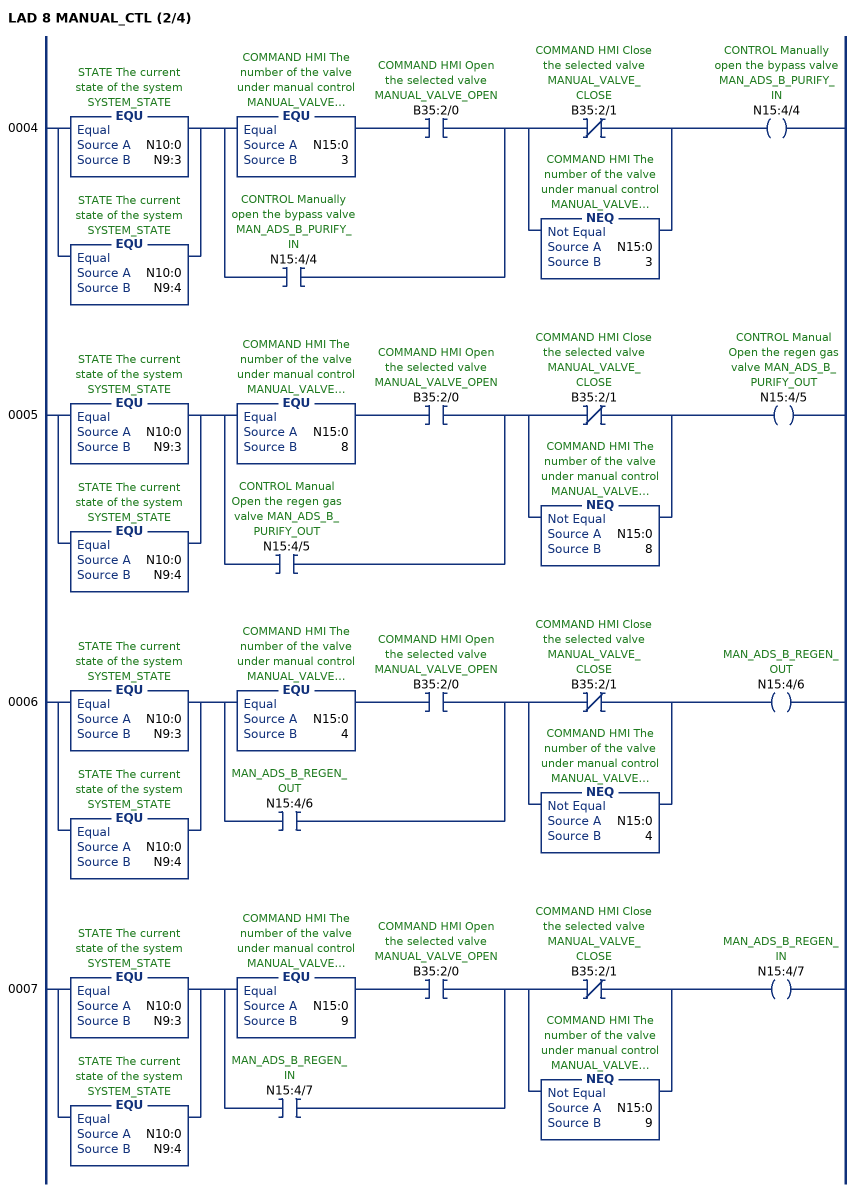
% Rung: 4 %
SOR BST EQU N10:0 N9:3 NXB EQU N10:0 N9:4 BND BST EQU N15:0 3 XIC B35:2/0 NXB XIC N15:4/4 BND BST XIO B35:2/1 NXB NEQ N15:0 3 BND OTE N15:4/4 EOR
%   N10:0  SYSTEM_STATE  "STATE The current state of the system" %
%   N9:3  SYSTEM_MANUAL  "STATE System Manual" %
%   N9:4  SYSTEM_ALARM  "STATE System Alarm" %
%   N15:0  MANUAL_VALVE_NUMBER  "COMMAND HMI The number of the valve under manual control" %
%   B35:2/0  MANUAL_VALVE_OPEN  "COMMAND HMI Open the selected valve" %
%   N15:4/4  MAN_ADS_B_PURIFY_IN  "CONTROL Manually open the bypass valve" %
%   B35:2/1  MANUAL_VALVE_CLOSE  "COMMAND HMI Close the selected valve" %
% Rung: 5 %
SOR BST EQU N10:0 N9:3 NXB EQU N10:0 N9:4 BND BST EQU N15:0 8 XIC B35:2/0 NXB XIC N15:4/5 BND BST XIO B35:2/1 NXB NEQ N15:0 8 BND OTE N15:4/5 EOR
%   N10:0  SYSTEM_STATE  "STATE The current state of the system" %
%   N9:3  SYSTEM_MANUAL  "STATE System Manual" %
%   N9:4  SYSTEM_ALARM  "STATE System Alarm" %
%   N15:0  MANUAL_VALVE_NUMBER  "COMMAND HMI The number of the valve under manual control" %
%   B35:2/0  MANUAL_VALVE_OPEN  "COMMAND HMI Open the selected valve" %
%   N15:4/5  MAN_ADS_B_PURIFY_OUT  "CONTROL Manual Open the regen gas valve" %
%   B35:2/1  MANUAL_VALVE_CLOSE  "COMMAND HMI Close the selected valve" %
% Rung: 6 %
SOR BST EQU N10:0 N9:3 NXB EQU N10:0 N9:4 BND BST EQU N15:0 4 XIC B35:2/0 NXB XIC N15:4/6 BND BST XIO B35:2/1 NXB NEQ N15:0 4 BND OTE N15:4/6 EOR
%   N10:0  SYSTEM_STATE  "STATE The current state of the system" %
%   N9:3  SYSTEM_MANUAL  "STATE System Manual" %
%   N9:4  SYSTEM_ALARM  "STATE System Alarm" %
%   N15:0  MANUAL_VALVE_NUMBER  "COMMAND HMI The number of the valve under manual control" %
%   B35:2/0  MANUAL_VALVE_OPEN  "COMMAND HMI Open the selected valve" %
%   N15:4/6  MAN_ADS_B_REGEN_OUT %
%   B35:2/1  MANUAL_VALVE_CLOSE  "COMMAND HMI Close the selected valve" %
% Rung: 7 %
SOR BST EQU N10:0 N9:3 NXB EQU N10:0 N9:4 BND BST EQU N15:0 9 XIC B35:2/0 NXB XIC N15:4/7 BND BST XIO B35:2/1 NXB NEQ N15:0 9 BND OTE N15:4/7 EOR
%   N10:0  SYSTEM_STATE  "STATE The current state of the system" %
%   N9:3  SYSTEM_MANUAL  "STATE System Manual" %
%   N9:4  SYSTEM_ALARM  "STATE System Alarm" %
%   N15:0  MANUAL_VALVE_NUMBER  "COMMAND HMI The number of the valve under manual control" %
%   B35:2/0  MANUAL_VALVE_OPEN  "COMMAND HMI Open the selected valve" %
%   N15:4/7  MAN_ADS_B_REGEN_IN %
%   B35:2/1  MANUAL_VALVE_CLOSE  "COMMAND HMI Close the selected valve" %

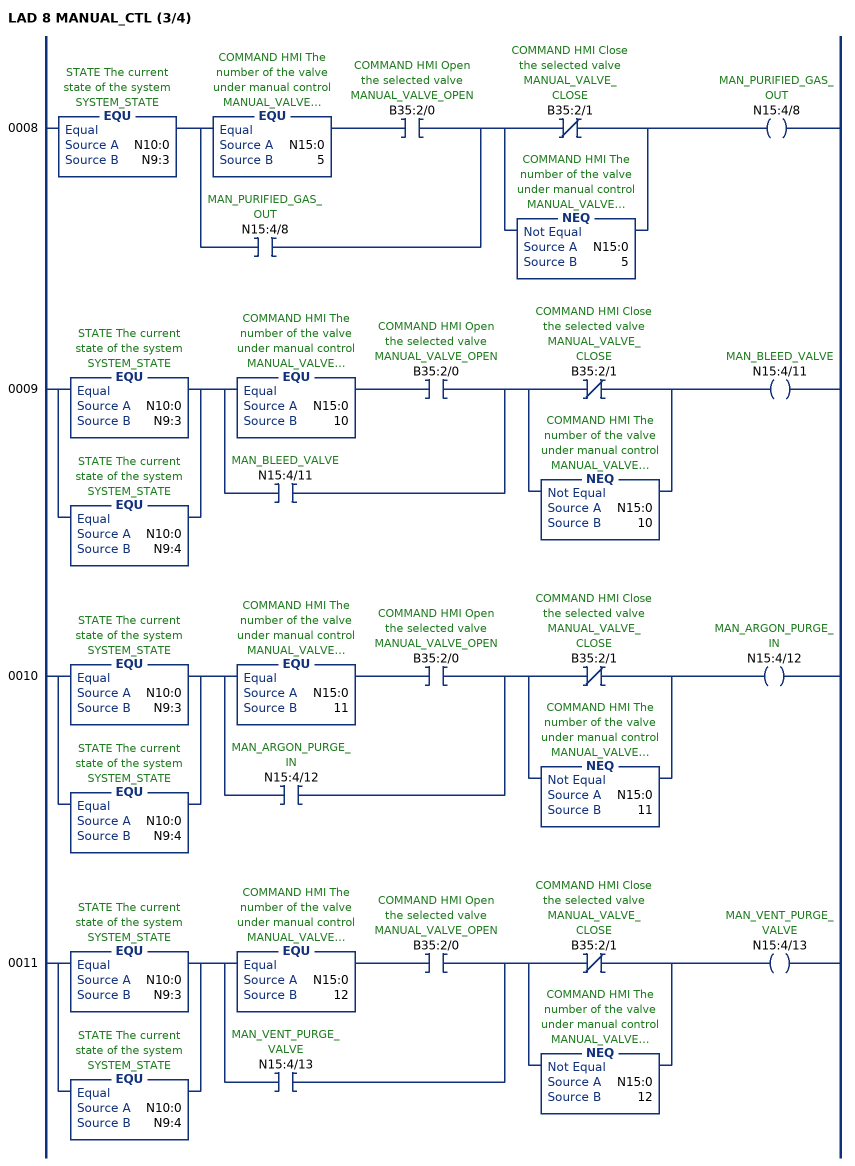
% Rung: 8 %
SOR EQU N10:0 N9:3 BST EQU N15:0 5 XIC B35:2/0 NXB XIC N15:4/8 BND BST XIO B35:2/1 NXB NEQ N15:0 5 BND OTE N15:4/8 EOR
%   N10:0  SYSTEM_STATE  "STATE The current state of the system" %
%   N9:3  SYSTEM_MANUAL  "STATE System Manual" %
%   N15:0  MANUAL_VALVE_NUMBER  "COMMAND HMI The number of the valve under manual control" %
%   B35:2/0  MANUAL_VALVE_OPEN  "COMMAND HMI Open the selected valve" %
%   N15:4/8  MAN_PURIFIED_GAS_OUT %
%   B35:2/1  MANUAL_VALVE_CLOSE  "COMMAND HMI Close the selected valve" %
% Rung: 9 %
SOR BST EQU N10:0 N9:3 NXB EQU N10:0 N9:4 BND BST EQU N15:0 10 XIC B35:2/0 NXB XIC N15:4/11 BND BST XIO B35:2/1 NXB NEQ N15:0 10 BND OTE N15:4/11 EOR
%   N10:0  SYSTEM_STATE  "STATE The current state of the system" %
%   N9:3  SYSTEM_MANUAL  "STATE System Manual" %
%   N9:4  SYSTEM_ALARM  "STATE System Alarm" %
%   N15:0  MANUAL_VALVE_NUMBER  "COMMAND HMI The number of the valve under manual control" %
%   B35:2/0  MANUAL_VALVE_OPEN  "COMMAND HMI Open the selected valve" %
%   N15:4/11  MAN_BLEED_VALVE %
%   B35:2/1  MANUAL_VALVE_CLOSE  "COMMAND HMI Close the selected valve" %
% Rung: 10 %
SOR BST EQU N10:0 N9:3 NXB EQU N10:0 N9:4 BND BST EQU N15:0 11 XIC B35:2/0 NXB XIC N15:4/12 BND BST XIO B35:2/1 NXB NEQ N15:0 11 BND OTE N15:4/12 EOR
%   N10:0  SYSTEM_STATE  "STATE The current state of the system" %
%   N9:3  SYSTEM_MANUAL  "STATE System Manual" %
%   N9:4  SYSTEM_ALARM  "STATE System Alarm" %
%   N15:0  MANUAL_VALVE_NUMBER  "COMMAND HMI The number of the valve under manual control" %
%   B35:2/0  MANUAL_VALVE_OPEN  "COMMAND HMI Open the selected valve" %
%   N15:4/12  MAN_ARGON_PURGE_IN %
%   B35:2/1  MANUAL_VALVE_CLOSE  "COMMAND HMI Close the selected valve" %
% Rung: 11 %
SOR BST EQU N10:0 N9:3 NXB EQU N10:0 N9:4 BND BST EQU N15:0 12 XIC B35:2/0 NXB XIC N15:4/13 BND BST XIO B35:2/1 NXB NEQ N15:0 12 BND OTE N15:4/13 EOR
%   N10:0  SYSTEM_STATE  "STATE The current state of the system" %
%   N9:3  SYSTEM_MANUAL  "STATE System Manual" %
%   N9:4  SYSTEM_ALARM  "STATE System Alarm" %
%   N15:0  MANUAL_VALVE_NUMBER  "COMMAND HMI The number of the valve under manual control" %
%   B35:2/0  MANUAL_VALVE_OPEN  "COMMAND HMI Open the selected valve" %
%   N15:4/13  MAN_VENT_PURGE_VALVE %
%   B35:2/1  MANUAL_VALVE_CLOSE  "COMMAND HMI Close the selected valve" %

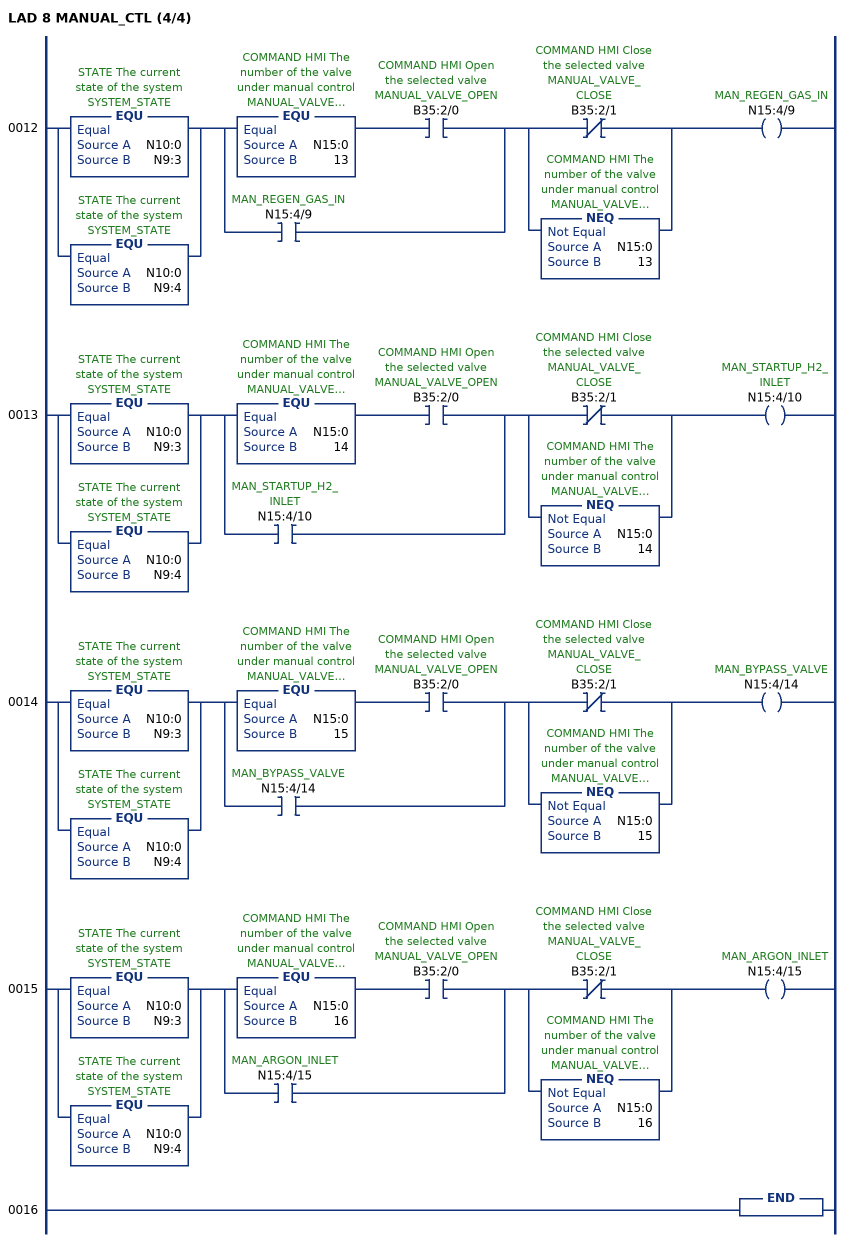
% Rung: 12 %
SOR BST EQU N10:0 N9:3 NXB EQU N10:0 N9:4 BND BST EQU N15:0 13 XIC B35:2/0 NXB XIC N15:4/9 BND BST XIO B35:2/1 NXB NEQ N15:0 13 BND OTE N15:4/9 EOR
%   N10:0  SYSTEM_STATE  "STATE The current state of the system" %
%   N9:3  SYSTEM_MANUAL  "STATE System Manual" %
%   N9:4  SYSTEM_ALARM  "STATE System Alarm" %
%   N15:0  MANUAL_VALVE_NUMBER  "COMMAND HMI The number of the valve under manual control" %
%   B35:2/0  MANUAL_VALVE_OPEN  "COMMAND HMI Open the selected valve" %
%   N15:4/9  MAN_REGEN_GAS_IN %
%   B35:2/1  MANUAL_VALVE_CLOSE  "COMMAND HMI Close the selected valve" %
% Rung: 13 %
SOR BST EQU N10:0 N9:3 NXB EQU N10:0 N9:4 BND BST EQU N15:0 14 XIC B35:2/0 NXB XIC N15:4/10 BND BST XIO B35:2/1 NXB NEQ N15:0 14 BND OTE N15:4/10 EOR
%   N10:0  SYSTEM_STATE  "STATE The current state of the system" %
%   N9:3  SYSTEM_MANUAL  "STATE System Manual" %
%   N9:4  SYSTEM_ALARM  "STATE System Alarm" %
%   N15:0  MANUAL_VALVE_NUMBER  "COMMAND HMI The number of the valve under manual control" %
%   B35:2/0  MANUAL_VALVE_OPEN  "COMMAND HMI Open the selected valve" %
%   N15:4/10  MAN_STARTUP_H2_INLET %
%   B35:2/1  MANUAL_VALVE_CLOSE  "COMMAND HMI Close the selected valve" %
% Rung: 14 %
SOR BST EQU N10:0 N9:3 NXB EQU N10:0 N9:4 BND BST EQU N15:0 15 XIC B35:2/0 NXB XIC N15:4/14 BND BST XIO B35:2/1 NXB NEQ N15:0 15 BND OTE N15:4/14 EOR
%   N10:0  SYSTEM_STATE  "STATE The current state of the system" %
%   N9:3  SYSTEM_MANUAL  "STATE System Manual" %
%   N9:4  SYSTEM_ALARM  "STATE System Alarm" %
%   N15:0  MANUAL_VALVE_NUMBER  "COMMAND HMI The number of the valve under manual control" %
%   B35:2/0  MANUAL_VALVE_OPEN  "COMMAND HMI Open the selected valve" %
%   N15:4/14  MAN_BYPASS_VALVE %
%   B35:2/1  MANUAL_VALVE_CLOSE  "COMMAND HMI Close the selected valve" %
% Rung: 15 %
SOR BST EQU N10:0 N9:3 NXB EQU N10:0 N9:4 BND BST EQU N15:0 16 XIC B35:2/0 NXB XIC N15:4/15 BND BST XIO B35:2/1 NXB NEQ N15:0 16 BND OTE N15:4/15 EOR
%   N10:0  SYSTEM_STATE  "STATE The current state of the system" %
%   N9:3  SYSTEM_MANUAL  "STATE System Manual" %
%   N9:4  SYSTEM_ALARM  "STATE System Alarm" %
%   N15:0  MANUAL_VALVE_NUMBER  "COMMAND HMI The number of the valve under manual control" %
%   B35:2/0  MANUAL_VALVE_OPEN  "COMMAND HMI Open the selected valve" %
%   N15:4/15  MAN_ARGON_INLET %
%   B35:2/1  MANUAL_VALVE_CLOSE  "COMMAND HMI Close the selected valve" %
% Rung: 16 %
SOR END EOR

LADDER 9 "STARTUP"
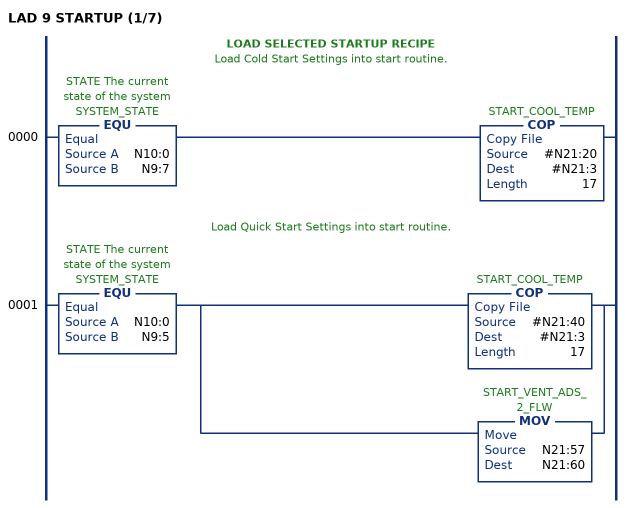
% Rung: 0 %
% TITLE: LOAD SELECTED STARTUP RECIPE %
% Load Cold Start Settings into start routine. %
SOR EQU N10:0 N9:7 COP #N21:20 #N21:3 17 EOR
%   N10:0  SYSTEM_STATE  "STATE The current state of the system" %
%   N9:7  SYSTEM_COLD_START %
%   N21:20  COLD_COOL_TEMP %
%   N21:3  START_COOL_TEMP %
% Rung: 1 %
% Load Quick Start Settings into start routine. %
SOR EQU N10:0 N9:5 BST COP #N21:40 #N21:3 17 NXB MOV N21:57 N21:60 BND EOR
%   N10:0  SYSTEM_STATE  "STATE The current state of the system" %
%   N9:5  SYSTEM_QUICK_START %
%   N21:40  QUICK_COOL_TEMP %
%   N21:3  START_COOL_TEMP %
%   N21:57  QUICK_VENT_ADS_2_FLW %
%   N21:60  START_VENT_ADS_2_FLW %

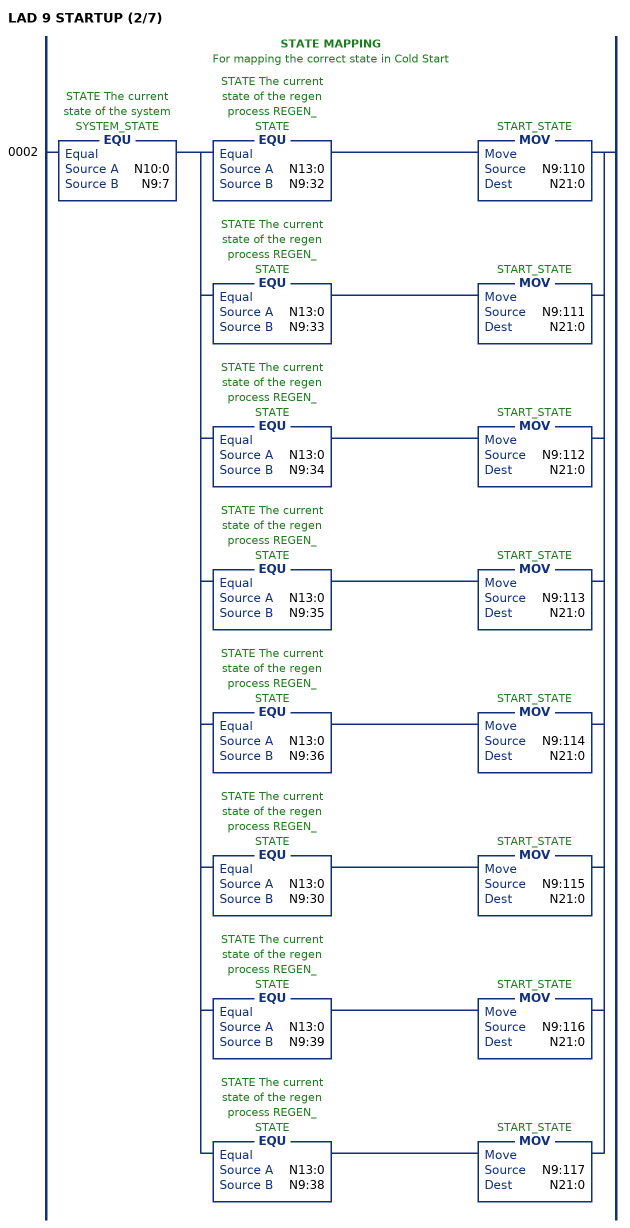
% Rung: 2 %
% TITLE: STATE MAPPING %
% For mapping the correct state in Cold Start %
SOR EQU N10:0 N9:7 BST EQU N13:0 N9:32 MOV N9:110 N21:0 NXB EQU N13:0 N9:33 MOV N9:111 N21:0 NXB EQU N13:0 N9:34 MOV N9:112 N21:0 NXB EQU N13:0 N9:35 MOV N9:113 N21:0 NXB EQU N13:0 N9:36 MOV N9:114 N21:0 NXB EQU N13:0 N9:30 MOV N9:115 N21:0 NXB EQU N13:0 N9:39 MOV N9:116 N21:0 NXB EQU N13:0 N9:38 MOV N9:117 N21:0 BND EOR
%   N10:0  SYSTEM_STATE  "STATE The current state of the system" %
%   N9:7  SYSTEM_COLD_START %
%   N13:0  REGEN_STATE  "STATE The current state of the regen process" %
%   N9:32  REGEN_VENT  "STATE Regen Vent" %
%   N9:110  START_REG_VENT %
%   N21:0  START_STATE %
%   N9:33  REGEN_HEAT_BED  "STATE Regen Heat wall" %
%   N9:111  START_REG_HEAT %
%   N9:34  REGEN_RUN  "STATE Regen Running" %
%   N9:112  START_REG_RUN %
%   N9:35  REGEN_COOL_WALL  "STATE Regen Cool wall" %
%   N9:113  START_REG_COOL %
%   N9:36  REGEN_COOL  "STATE Regen Cool" %
%   N9:114  START_REG_TIMED_COOL %
%   N9:30  REGEN_STANDBY  "STATE Regen Standby" %
%   N9:115  START_REG_STANDBY %
%   N9:39  REGEN_BACKFILL %
%   N9:116  START_REG_BACKFILL %
%   N9:38  REGEN_DONE %
%   N9:117  START_REG_DONE %

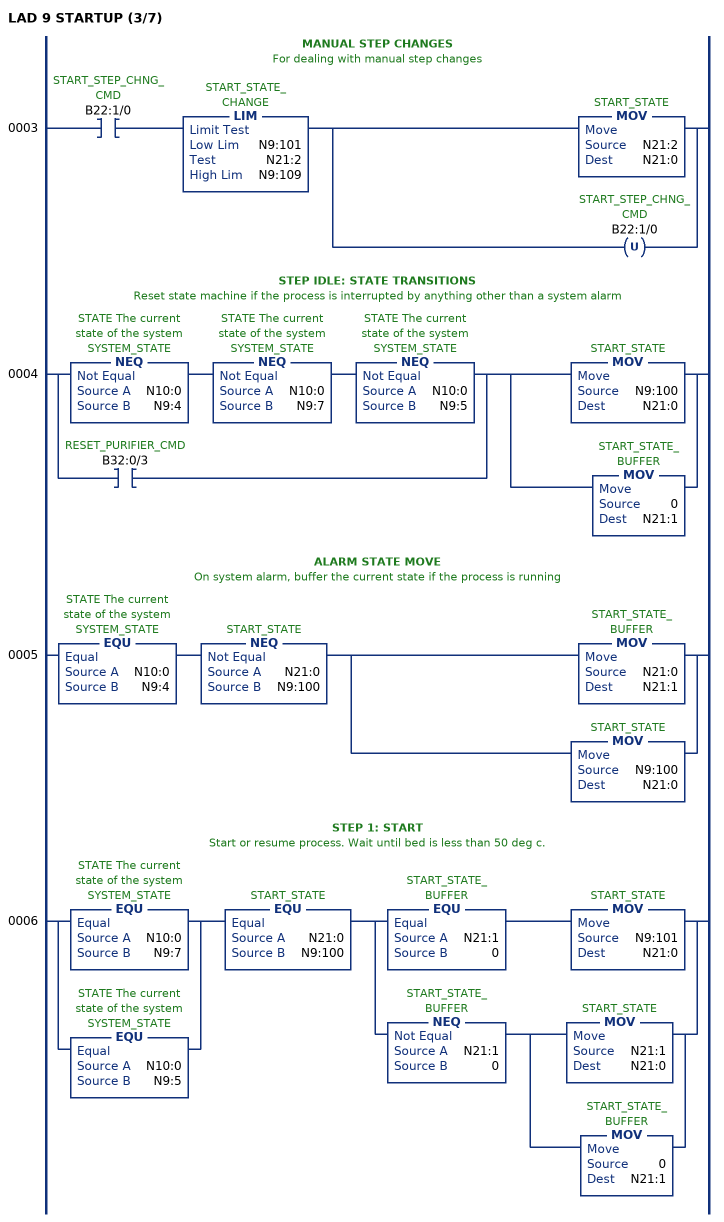
% Rung: 3 %
% TITLE: MANUAL STEP CHANGES %
% For dealing with manual step changes %
SOR XIC B22:1/0 LIM N9:101 N21:2 N9:109 BST MOV N21:2 N21:0 NXB OTU B22:1/0 BND EOR
%   B22:1/0  START_STEP_CHNG_CMD %
%   N9:101  START_COOL %
%   N21:2  START_STATE_CHANGE %
%   N9:109  START_BKFL_2 %
%   N21:0  START_STATE %
% Rung: 4 %
% TITLE: STEP IDLE: STATE TRANSITIONS %
% Reset state machine if the process is interrupted by anything other than a system alarm %
SOR BST NEQ N10:0 N9:4 NEQ N10:0 N9:7 NEQ N10:0 N9:5 NXB XIC B32:0/3 BND BST MOV N9:100 N21:0 NXB MOV 0 N21:1 BND EOR
%   N10:0  SYSTEM_STATE  "STATE The current state of the system" %
%   N9:4  SYSTEM_ALARM  "STATE System Alarm" %
%   N9:7  SYSTEM_COLD_START %
%   N9:5  SYSTEM_QUICK_START %
%   B32:0/3  RESET_PURIFIER_CMD %
%   N9:100  START_IDLE %
%   N21:0  START_STATE %
%   N21:1  START_STATE_BUFFER %
% Rung: 5 %
% TITLE: ALARM STATE MOVE %
% On system alarm, buffer the current state if the process is running %
SOR EQU N10:0 N9:4 NEQ N21:0 N9:100 BST MOV N21:0 N21:1 NXB MOV N9:100 N21:0 BND EOR
%   N10:0  SYSTEM_STATE  "STATE The current state of the system" %
%   N9:4  SYSTEM_ALARM  "STATE System Alarm" %
%   N21:0  START_STATE %
%   N9:100  START_IDLE %
%   N21:1  START_STATE_BUFFER %
% Rung: 6 %
% TITLE: STEP 1: START %
% Start or resume process. Wait until bed is less than 50 deg c. %
SOR BST EQU N10:0 N9:7 NXB EQU N10:0 N9:5 BND EQU N21:0 N9:100 BST EQU N21:1 0 MOV N9:101 N21:0 NXB NEQ N21:1 0 BST MOV N21:1 N21:0 NXB MOV 0 N21:1 BND BND EOR
%   N10:0  SYSTEM_STATE  "STATE The current state of the system" %
%   N9:7  SYSTEM_COLD_START %
%   N9:5  SYSTEM_QUICK_START %
%   N21:0  START_STATE %
%   N9:100  START_IDLE %
%   N21:1  START_STATE_BUFFER %
%   N9:101  START_COOL %

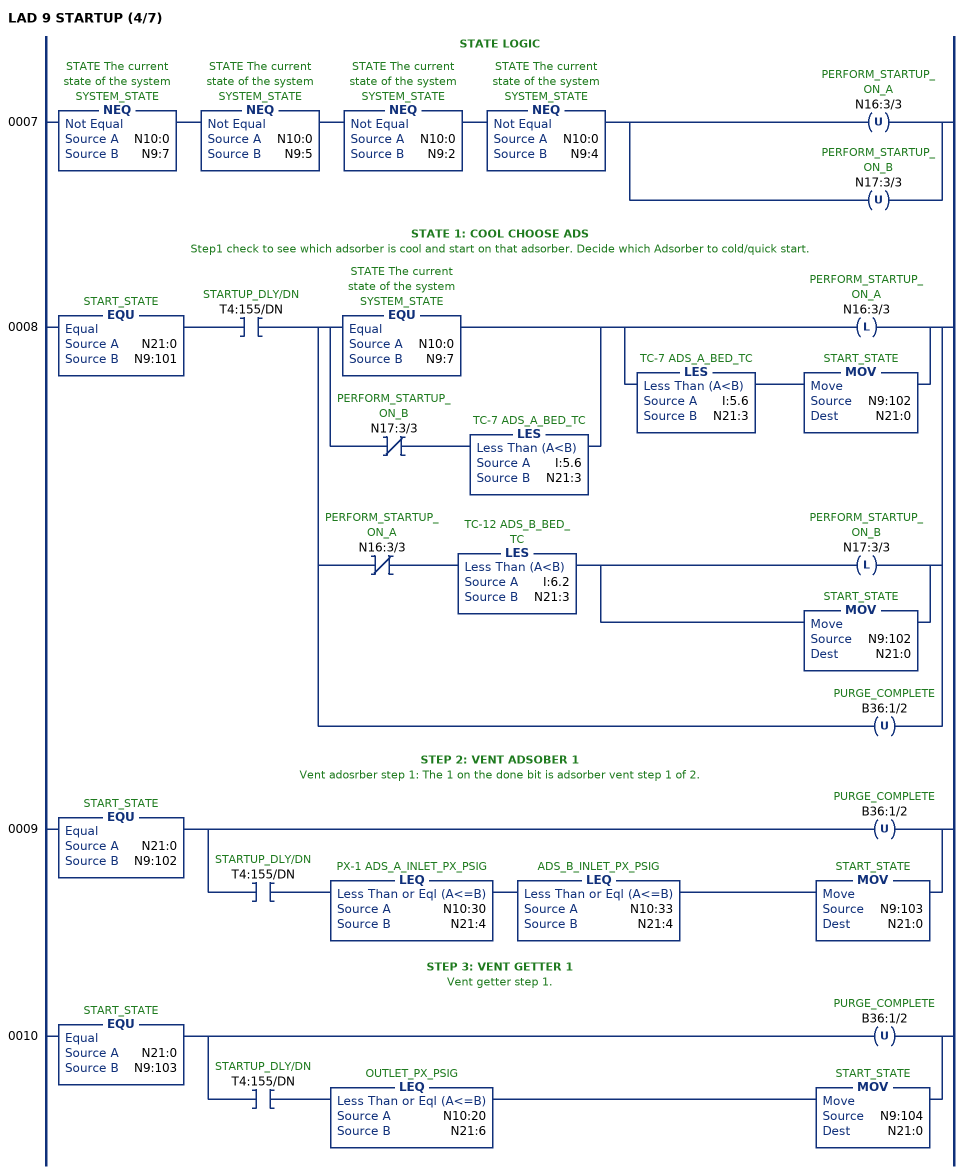
% Rung: 7 %
% TITLE: STATE LOGIC %
SOR NEQ N10:0 N9:7 NEQ N10:0 N9:5 NEQ N10:0 N9:2 NEQ N10:0 N9:4 BST OTU N16:3/3 NXB OTU N17:3/3 BND EOR
%   N10:0  SYSTEM_STATE  "STATE The current state of the system" %
%   N9:7  SYSTEM_COLD_START %
%   N9:5  SYSTEM_QUICK_START %
%   N9:2  SYSTEM_PROCESS  "STATE System Process" %
%   N9:4  SYSTEM_ALARM  "STATE System Alarm" %
%   N16:3/3  PERFORM_STARTUP_ON_A %
%   N17:3/3  PERFORM_STARTUP_ON_B %
% Rung: 8 %
% TITLE: STATE 1: COOL CHOOSE ADS %
% Step1 check to see which adsorber is cool and start on that adsorber. Decide which Adsorber to cold/quick start. %
SOR EQU N21:0 N9:101 XIC T4:155/DN BST BST EQU N10:0 N9:7 NXB XIO N17:3/3 LES I:5.6 N21:3 BND BST OTL N16:3/3 NXB LES I:5.6 N21:3 MOV N9:102 N21:0 BND NXB XIO N16:3/3 LES I:6.2 N21:3 BST OTL N17:3/3 NXB MOV N9:102 N21:0 BND NXB OTU B36:1/2 BND EOR
%   N21:0  START_STATE %
%   N9:101  START_COOL %
%   T4:155  STARTUP_DLY %
%   N10:0  SYSTEM_STATE  "STATE The current state of the system" %
%   N9:7  SYSTEM_COLD_START %
%   N17:3/3  PERFORM_STARTUP_ON_B %
%   I:5.6  ADS_A_BED_TC  "TC-7" %
%   N21:3  START_COOL_TEMP %
%   N16:3/3  PERFORM_STARTUP_ON_A %
%   N9:102  START_VENT_ADS_1 %
%   I:6.2  ADS_B_BED_TC  "TC-12" %
%   B36:1/2  PURGE_COMPLETE %
% Rung: 9 %
% TITLE: STEP 2: VENT ADSOBER 1 %
% Vent adosrber step 1: The 1 on the done bit is adsorber vent step 1 of 2. %
SOR EQU N21:0 N9:102 BST OTU B36:1/2 NXB XIC T4:155/DN LEQ N10:30 N21:4 LEQ N10:33 N21:4 MOV N9:103 N21:0 BND EOR
%   N21:0  START_STATE %
%   N9:102  START_VENT_ADS_1 %
%   B36:1/2  PURGE_COMPLETE %
%   T4:155  STARTUP_DLY %
%   N10:30  ADS_A_INLET_PX_PSIG  "PX-1" %
%   N21:4  START_VENT_ADS_1_PRS %
%   N10:33  ADS_B_INLET_PX_PSIG %
%   N9:103  START_VENT_GET_1 %
% Rung: 10 %
% TITLE: STEP 3: VENT GETTER 1 %
% Vent getter step 1. %
SOR EQU N21:0 N9:103 BST OTU B36:1/2 NXB XIC T4:155/DN LEQ N10:20 N21:6 MOV N9:104 N21:0 BND EOR
%   N21:0  START_STATE %
%   N9:103  START_VENT_GET_1 %
%   B36:1/2  PURGE_COMPLETE %
%   T4:155  STARTUP_DLY %
%   N10:20  OUTLET_PX_PSIG %
%   N21:6  START_VENT_GET_1_PRS %
%   N9:104  START_HEAT_GETTER %

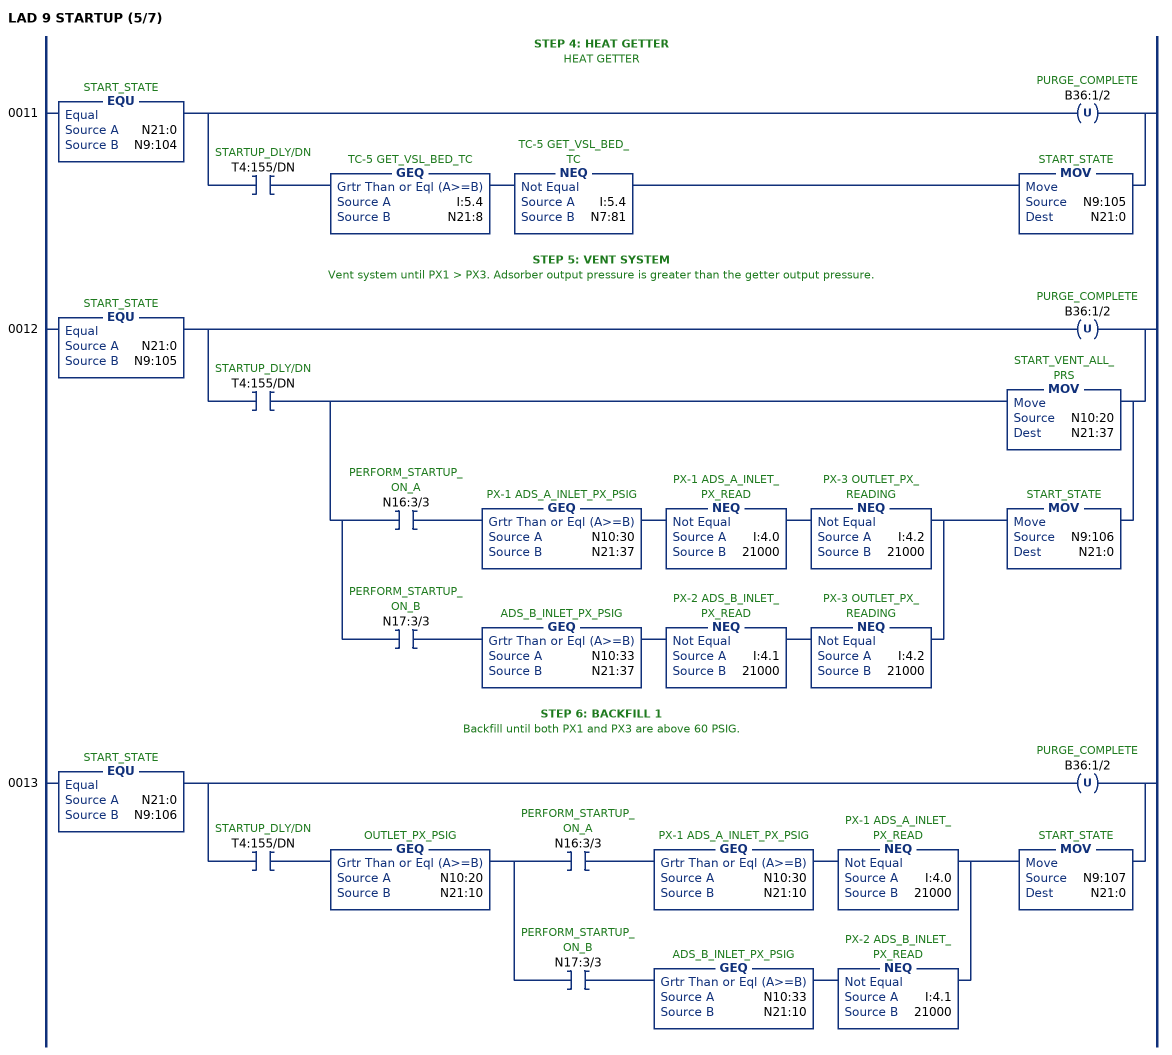
% Rung: 11 %
% TITLE: STEP 4: HEAT GETTER %
% HEAT GETTER %
SOR EQU N21:0 N9:104 BST OTU B36:1/2 NXB XIC T4:155/DN GEQ I:5.4 N21:8 NEQ I:5.4 N7:81 MOV N9:105 N21:0 BND EOR
%   N21:0  START_STATE %
%   N9:104  START_HEAT_GETTER %
%   B36:1/2  PURGE_COMPLETE %
%   T4:155  STARTUP_DLY %
%   I:5.4  GET_VSL_BED_TC  "TC-5" %
%   N21:8  START_HEAT_TEMP %
%   N7:81  TC_OPEN_SP  "CONFIG The value read by an open TC input" %
%   N9:105  START_VENT_ALL %
% Rung: 12 %
% TITLE: STEP 5: VENT SYSTEM %
% Vent system until PX1 > PX3. Adsorber output pressure is greater than the getter output pressure. %
SOR EQU N21:0 N9:105 BST OTU B36:1/2 NXB XIC T4:155/DN BST MOV N10:20 N21:37 NXB BST XIC N16:3/3 GEQ N10:30 N21:37 NEQ I:4.0 21000 NEQ I:4.2 21000 NXB XIC N17:3/3 GEQ N10:33 N21:37 NEQ I:4.1 21000 NEQ I:4.2 21000 BND MOV N9:106 N21:0 BND BND EOR
%   N21:0  START_STATE %
%   N9:105  START_VENT_ALL %
%   B36:1/2  PURGE_COMPLETE %
%   T4:155  STARTUP_DLY %
%   N10:20  OUTLET_PX_PSIG %
%   N21:37  START_VENT_ALL_PRS %
%   N16:3/3  PERFORM_STARTUP_ON_A %
%   N10:30  ADS_A_INLET_PX_PSIG  "PX-1" %
%   I:4.0  ADS_A_INLET_PX_READ  "PX-1" %
%   I:4.2  OUTLET_PX_READING  "PX-3" %
%   N17:3/3  PERFORM_STARTUP_ON_B %
%   N10:33  ADS_B_INLET_PX_PSIG %
%   I:4.1  ADS_B_INLET_PX_READ  "PX-2" %
%   N9:106  START_BACKFILL_1 %
% Rung: 13 %
% TITLE: STEP 6: BACKFILL 1 %
% Backfill until both PX1 and PX3 are above 60 PSIG. %
SOR EQU N21:0 N9:106 BST OTU B36:1/2 NXB XIC T4:155/DN GEQ N10:20 N21:10 BST XIC N16:3/3 GEQ N10:30 N21:10 NEQ I:4.0 21000 NXB XIC N17:3/3 GEQ N10:33 N21:10 NEQ I:4.1 21000 BND MOV N9:107 N21:0 BND EOR
%   N21:0  START_STATE %
%   N9:106  START_BACKFILL_1 %
%   B36:1/2  PURGE_COMPLETE %
%   T4:155  STARTUP_DLY %
%   N10:20  OUTLET_PX_PSIG %
%   N21:10  START_BKFIL_1_PRS %
%   N16:3/3  PERFORM_STARTUP_ON_A %
%   N10:30  ADS_A_INLET_PX_PSIG  "PX-1" %
%   I:4.0  ADS_A_INLET_PX_READ  "PX-1" %
%   N17:3/3  PERFORM_STARTUP_ON_B %
%   N10:33  ADS_B_INLET_PX_PSIG %
%   I:4.1  ADS_B_INLET_PX_READ  "PX-2" %
%   N9:107  START_VENT_ADS_2 %

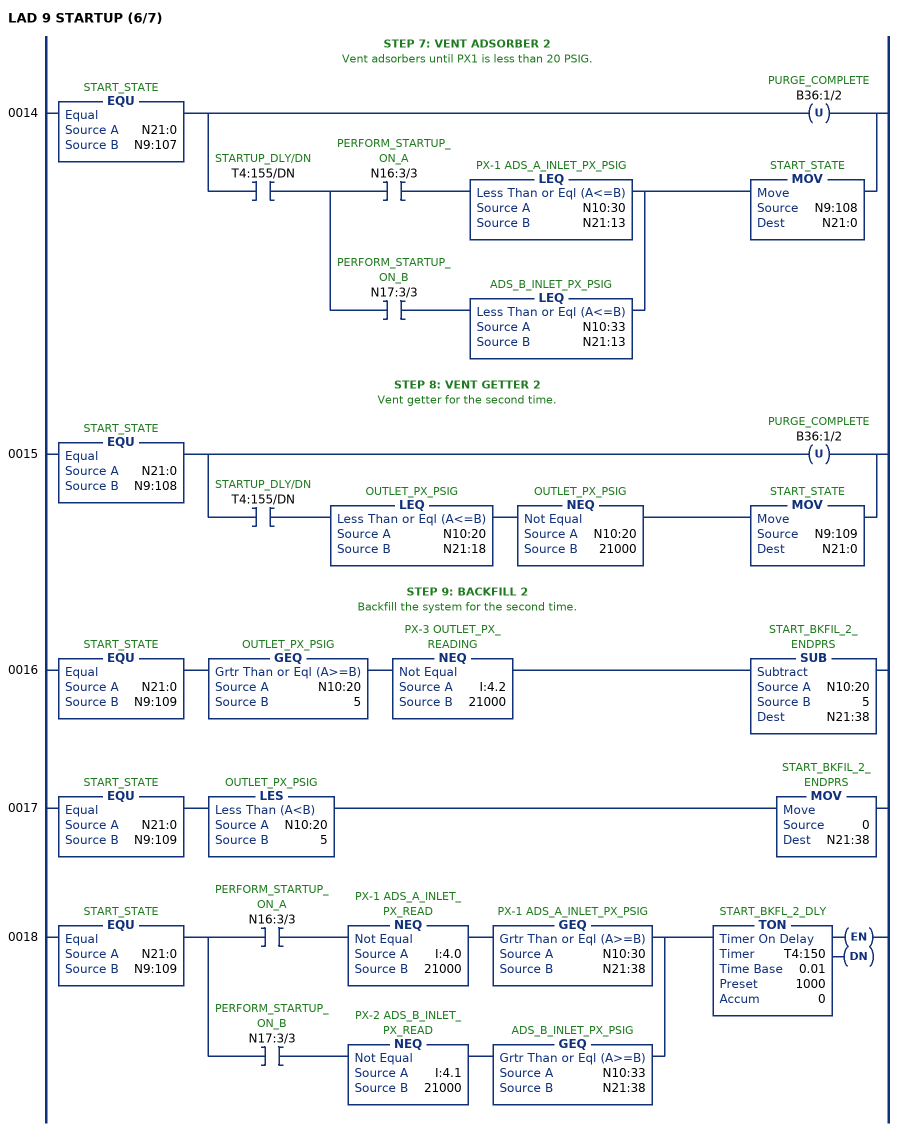
% Rung: 14 %
% TITLE: STEP 7: VENT ADSORBER 2 %
% Vent adsorbers until PX1 is less than 20 PSIG. %
SOR EQU N21:0 N9:107 BST OTU B36:1/2 NXB XIC T4:155/DN BST XIC N16:3/3 LEQ N10:30 N21:13 NXB XIC N17:3/3 LEQ N10:33 N21:13 BND MOV N9:108 N21:0 BND EOR
%   N21:0  START_STATE %
%   N9:107  START_VENT_ADS_2 %
%   B36:1/2  PURGE_COMPLETE %
%   T4:155  STARTUP_DLY %
%   N16:3/3  PERFORM_STARTUP_ON_A %
%   N10:30  ADS_A_INLET_PX_PSIG  "PX-1" %
%   N21:13  START_VENT_ADS_2_PRS %
%   N17:3/3  PERFORM_STARTUP_ON_B %
%   N10:33  ADS_B_INLET_PX_PSIG %
%   N9:108  START_VENT_GET_2 %
% Rung: 15 %
% TITLE: STEP 8: VENT GETTER 2 %
% Vent getter for the second time. %
SOR EQU N21:0 N9:108 BST OTU B36:1/2 NXB XIC T4:155/DN LEQ N10:20 N21:18 NEQ N10:20 21000 MOV N9:109 N21:0 BND EOR
%   N21:0  START_STATE %
%   N9:108  START_VENT_GET_2 %
%   B36:1/2  PURGE_COMPLETE %
%   T4:155  STARTUP_DLY %
%   N10:20  OUTLET_PX_PSIG %
%   N21:18  START_VENT_GET_2_PRS %
%   N9:109  START_BKFL_2 %
% Rung: 16 %
% TITLE: STEP 9: BACKFILL 2 %
% Backfill the system for the second time. %
SOR EQU N21:0 N9:109 GEQ N10:20 5 NEQ I:4.2 21000 SUB N10:20 5 N21:38 EOR
%   N21:0  START_STATE %
%   N9:109  START_BKFL_2 %
%   N10:20  OUTLET_PX_PSIG %
%   I:4.2  OUTLET_PX_READING  "PX-3" %
%   N21:38  START_BKFIL_2_ENDPRS %
% Rung: 17 %
SOR EQU N21:0 N9:109 LES N10:20 5 MOV 0 N21:38 EOR
%   N21:0  START_STATE %
%   N9:109  START_BKFL_2 %
%   N10:20  OUTLET_PX_PSIG %
%   N21:38  START_BKFIL_2_ENDPRS %
% Rung: 18 %
SOR EQU N21:0 N9:109 BST XIC N16:3/3 NEQ I:4.0 21000 GEQ N10:30 N21:38 NXB XIC N17:3/3 NEQ I:4.1 21000 GEQ N10:33 N21:38 BND TON T4:150 0.01 1000 0 EOR
%   N21:0  START_STATE %
%   N9:109  START_BKFL_2 %
%   N16:3/3  PERFORM_STARTUP_ON_A %
%   I:4.0  ADS_A_INLET_PX_READ  "PX-1" %
%   N10:30  ADS_A_INLET_PX_PSIG  "PX-1" %
%   N21:38  START_BKFIL_2_ENDPRS %
%   N17:3/3  PERFORM_STARTUP_ON_B %
%   I:4.1  ADS_B_INLET_PX_READ  "PX-2" %
%   N10:33  ADS_B_INLET_PX_PSIG %
%   T4:150  START_BKFL_2_DLY %

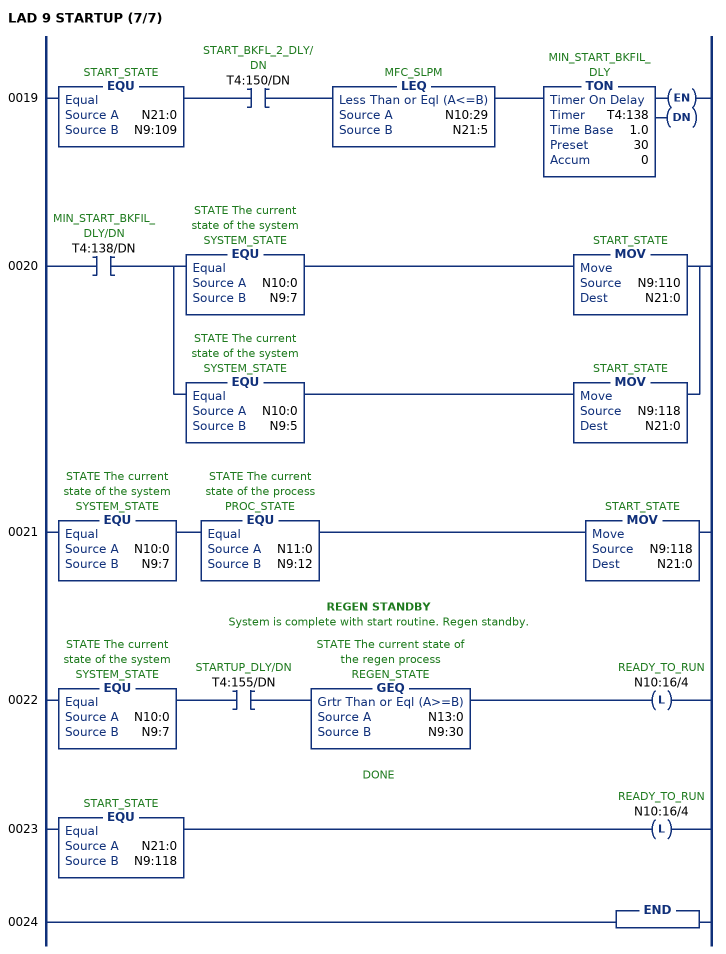
% Rung: 19 %
SOR EQU N21:0 N9:109 XIC T4:150/DN LEQ N10:29 N21:5 TON T4:138 1.0 30 0 EOR
%   N21:0  START_STATE %
%   N9:109  START_BKFL_2 %
%   T4:150  START_BKFL_2_DLY %
%   N10:29  MFC_SLPM %
%   N21:5  START_BKFIL_2_END %
%   T4:138  MIN_START_BKFIL_DLY %
% Rung: 20 %
SOR XIC T4:138/DN BST EQU N10:0 N9:7 MOV N9:110 N21:0 NXB EQU N10:0 N9:5 MOV N9:118 N21:0 BND EOR
%   T4:138  MIN_START_BKFIL_DLY %
%   N10:0  SYSTEM_STATE  "STATE The current state of the system" %
%   N9:7  SYSTEM_COLD_START %
%   N9:110  START_REG_VENT %
%   N21:0  START_STATE %
%   N9:5  SYSTEM_QUICK_START %
%   N9:118  START_DONE %
% Rung: 21 %
SOR EQU N10:0 N9:7 EQU N11:0 N9:12 MOV N9:118 N21:0 EOR
%   N10:0  SYSTEM_STATE  "STATE The current state of the system" %
%   N9:7  SYSTEM_COLD_START %
%   N11:0  PROC_STATE  "STATE The current state of the process" %
%   N9:12  PROC_PFY_B_REG_A  "STATE Process Purify B" %
%   N9:118  START_DONE %
%   N21:0  START_STATE %
% Rung: 22 %
% TITLE: REGEN STANDBY %
% System is complete with start routine. Regen standby. %
SOR EQU N10:0 N9:7 XIC T4:155/DN GEQ N13:0 N9:30 OTL N10:16/4 EOR
%   N10:0  SYSTEM_STATE  "STATE The current state of the system" %
%   N9:7  SYSTEM_COLD_START %
%   T4:155  STARTUP_DLY %
%   N13:0  REGEN_STATE  "STATE The current state of the regen process" %
%   N9:30  REGEN_STANDBY  "STATE Regen Standby" %
%   N10:16/4  READY_TO_RUN %
% Rung: 23 %
% DONE %
SOR EQU N21:0 N9:118 OTL N10:16/4 EOR
%   N21:0  START_STATE %
%   N9:118  START_DONE %
%   N10:16/4  READY_TO_RUN %
% Rung: 24 %
SOR END EOR

LADDER 10 "PURIFY"    % Operates the purify control %
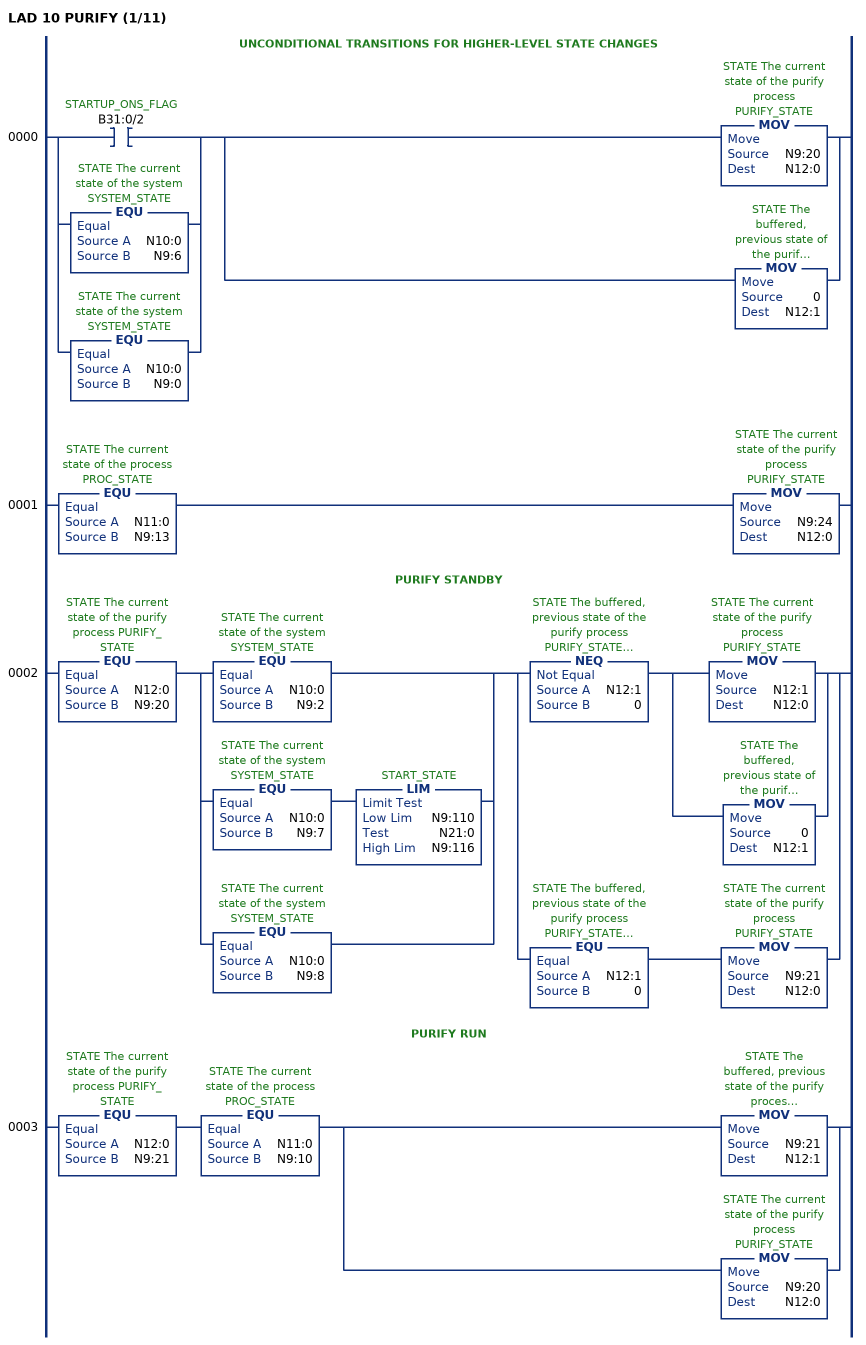
% Rung: 0 %
% TITLE: UNCONDITIONAL TRANSITIONS FOR HIGHER-LEVEL STATE CHANGES %
SOR BST XIC B31:0/2 NXB EQU N10:0 N9:6 NXB EQU N10:0 N9:0 BND BST MOV N9:20 N12:0 NXB MOV 0 N12:1 BND EOR
%   B31:0/2  STARTUP_ONS_FLAG %
%   N10:0  SYSTEM_STATE  "STATE The current state of the system" %
%   N9:6  SYSTEM_PURGE %
%   N9:0  SYSTEM_OFFLINE %
%   N9:20  PURIFY_STANDBY  "STATE Purify Standby" %
%   N12:0  PURIFY_STATE  "STATE The current state of the purify process" %
%   N12:1  PURIFY_STATE_BUFFER  "STATE The buffered, previous state of the purify process" %
% Rung: 1 %
SOR EQU N11:0 N9:13 MOV N9:24 N12:0 EOR
%   N11:0  PROC_STATE  "STATE The current state of the process" %
%   N9:13  PROC_OVERLAP  "STATE Process Purify Overlap" %
%   N9:24  PURIFY_OVERLAP  "STATE Puriify Overlap" %
%   N12:0  PURIFY_STATE  "STATE The current state of the purify process" %
% Rung: 2 %
% TITLE: PURIFY STANDBY %
SOR EQU N12:0 N9:20 BST EQU N10:0 N9:2 NXB EQU N10:0 N9:7 LIM N9:110 N21:0 N9:116 NXB EQU N10:0 N9:8 BND BST NEQ N12:1 0 BST MOV N12:1 N12:0 NXB MOV 0 N12:1 BND NXB EQU N12:1 0 MOV N9:21 N12:0 BND EOR
%   N12:0  PURIFY_STATE  "STATE The current state of the purify process" %
%   N9:20  PURIFY_STANDBY  "STATE Purify Standby" %
%   N10:0  SYSTEM_STATE  "STATE The current state of the system" %
%   N9:2  SYSTEM_PROCESS  "STATE System Process" %
%   N9:7  SYSTEM_COLD_START %
%   N9:110  START_REG_VENT %
%   N21:0  START_STATE %
%   N9:116  START_REG_BACKFILL %
%   N9:8  SYSTEM_SUPPLEMENTAL %
%   N12:1  PURIFY_STATE_BUFFER  "STATE The buffered, previous state of the purify process" %
%   N9:21  PURIFY_RUN  "STATE Purify running" %
% Rung: 3 %
% TITLE: PURIFY RUN %
SOR EQU N12:0 N9:21 EQU N11:0 N9:10 BST MOV N9:21 N12:1 NXB MOV N9:20 N12:0 BND EOR
%   N12:0  PURIFY_STATE  "STATE The current state of the purify process" %
%   N9:21  PURIFY_RUN  "STATE Purify running" %
%   N11:0  PROC_STATE  "STATE The current state of the process" %
%   N9:10  PROC_STANDBY  "STATE Process Standby" %
%   N12:1  PURIFY_STATE_BUFFER  "STATE The buffered, previous state of the purify process" %
%   N9:20  PURIFY_STANDBY  "STATE Purify Standby" %

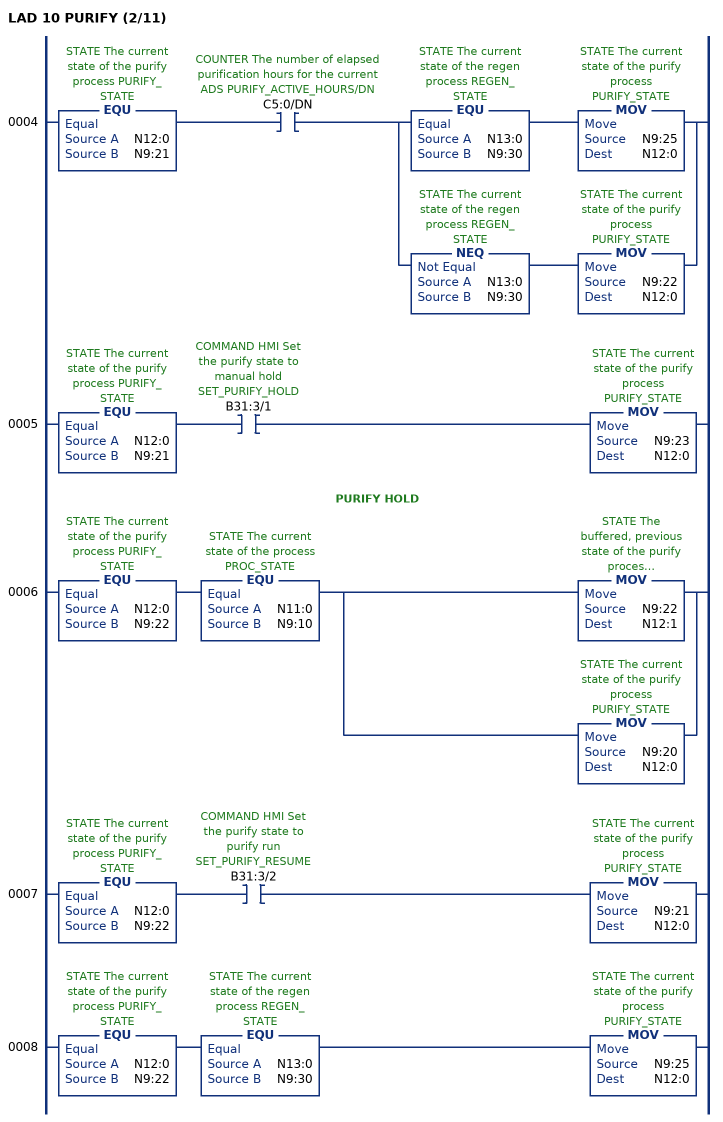
% Rung: 4 %
SOR EQU N12:0 N9:21 XIC C5:0/DN BST EQU N13:0 N9:30 MOV N9:25 N12:0 NXB NEQ N13:0 N9:30 MOV N9:22 N12:0 BND EOR
%   N12:0  PURIFY_STATE  "STATE The current state of the purify process" %
%   N9:21  PURIFY_RUN  "STATE Purify running" %
%   C5:0  PURIFY_ACTIVE_HOURS  "COUNTER The number of elapsed purification hours for the current ADS" %
%   N13:0  REGEN_STATE  "STATE The current state of the regen process" %
%   N9:30  REGEN_STANDBY  "STATE Regen Standby" %
%   N9:25  PURIFY_DONE %
%   N9:22  PURIFY_HOLD  "STATE Purify Hold" %
% Rung: 5 %
SOR EQU N12:0 N9:21 XIC B31:3/1 MOV N9:23 N12:0 EOR
%   N12:0  PURIFY_STATE  "STATE The current state of the purify process" %
%   N9:21  PURIFY_RUN  "STATE Purify running" %
%   B31:3/1  SET_PURIFY_HOLD  "COMMAND HMI Set the purify state to manual hold" %
%   N9:23  PURIFY_MANUAL_HOLD  "STATE Purify Manual Hold" %
% Rung: 6 %
% TITLE: PURIFY HOLD %
SOR EQU N12:0 N9:22 EQU N11:0 N9:10 BST MOV N9:22 N12:1 NXB MOV N9:20 N12:0 BND EOR
%   N12:0  PURIFY_STATE  "STATE The current state of the purify process" %
%   N9:22  PURIFY_HOLD  "STATE Purify Hold" %
%   N11:0  PROC_STATE  "STATE The current state of the process" %
%   N9:10  PROC_STANDBY  "STATE Process Standby" %
%   N12:1  PURIFY_STATE_BUFFER  "STATE The buffered, previous state of the purify process" %
%   N9:20  PURIFY_STANDBY  "STATE Purify Standby" %
% Rung: 7 %
SOR EQU N12:0 N9:22 XIC B31:3/2 MOV N9:21 N12:0 EOR
%   N12:0  PURIFY_STATE  "STATE The current state of the purify process" %
%   N9:22  PURIFY_HOLD  "STATE Purify Hold" %
%   B31:3/2  SET_PURIFY_RESUME  "COMMAND HMI Set the purify state to purify run" %
%   N9:21  PURIFY_RUN  "STATE Purify running" %
% Rung: 8 %
SOR EQU N12:0 N9:22 EQU N13:0 N9:30 MOV N9:25 N12:0 EOR
%   N12:0  PURIFY_STATE  "STATE The current state of the purify process" %
%   N9:22  PURIFY_HOLD  "STATE Purify Hold" %
%   N13:0  REGEN_STATE  "STATE The current state of the regen process" %
%   N9:30  REGEN_STANDBY  "STATE Regen Standby" %
%   N9:25  PURIFY_DONE %

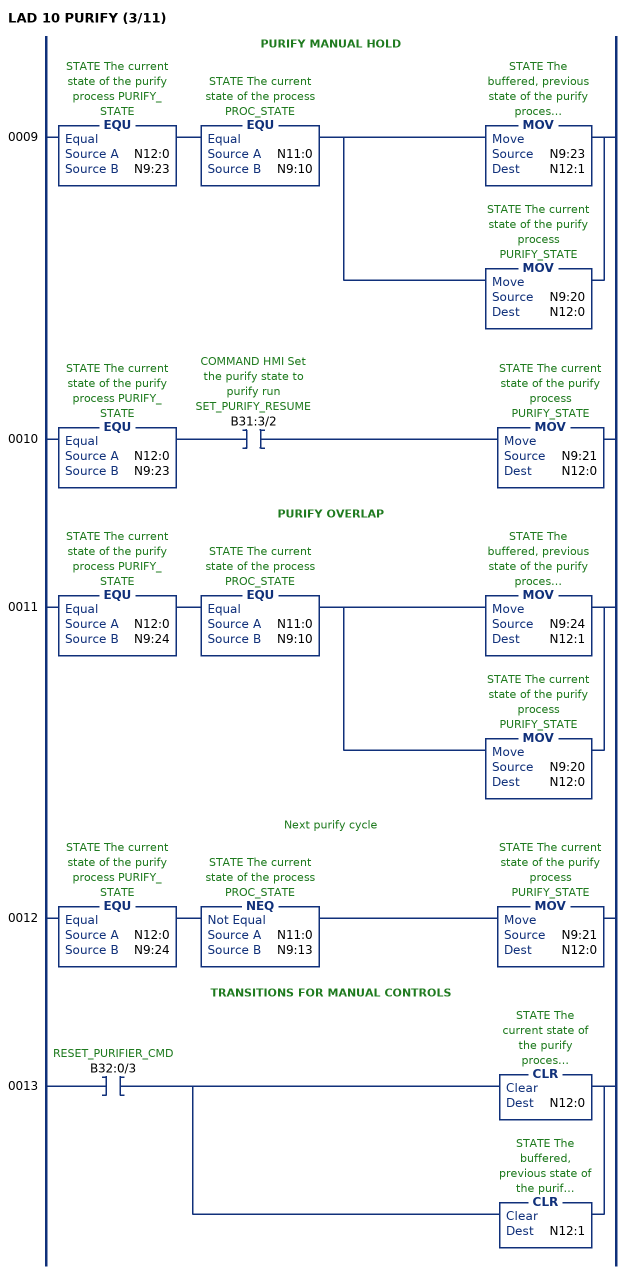
% Rung: 9 %
% TITLE: PURIFY MANUAL HOLD %
SOR EQU N12:0 N9:23 EQU N11:0 N9:10 BST MOV N9:23 N12:1 NXB MOV N9:20 N12:0 BND EOR
%   N12:0  PURIFY_STATE  "STATE The current state of the purify process" %
%   N9:23  PURIFY_MANUAL_HOLD  "STATE Purify Manual Hold" %
%   N11:0  PROC_STATE  "STATE The current state of the process" %
%   N9:10  PROC_STANDBY  "STATE Process Standby" %
%   N12:1  PURIFY_STATE_BUFFER  "STATE The buffered, previous state of the purify process" %
%   N9:20  PURIFY_STANDBY  "STATE Purify Standby" %
% Rung: 10 %
SOR EQU N12:0 N9:23 XIC B31:3/2 MOV N9:21 N12:0 EOR
%   N12:0  PURIFY_STATE  "STATE The current state of the purify process" %
%   N9:23  PURIFY_MANUAL_HOLD  "STATE Purify Manual Hold" %
%   B31:3/2  SET_PURIFY_RESUME  "COMMAND HMI Set the purify state to purify run" %
%   N9:21  PURIFY_RUN  "STATE Purify running" %
% Rung: 11 %
% TITLE: PURIFY OVERLAP %
SOR EQU N12:0 N9:24 EQU N11:0 N9:10 BST MOV N9:24 N12:1 NXB MOV N9:20 N12:0 BND EOR
%   N12:0  PURIFY_STATE  "STATE The current state of the purify process" %
%   N9:24  PURIFY_OVERLAP  "STATE Puriify Overlap" %
%   N11:0  PROC_STATE  "STATE The current state of the process" %
%   N9:10  PROC_STANDBY  "STATE Process Standby" %
%   N12:1  PURIFY_STATE_BUFFER  "STATE The buffered, previous state of the purify process" %
%   N9:20  PURIFY_STANDBY  "STATE Purify Standby" %
% Rung: 12 %
% Next purify cycle %
SOR EQU N12:0 N9:24 NEQ N11:0 N9:13 MOV N9:21 N12:0 EOR
%   N12:0  PURIFY_STATE  "STATE The current state of the purify process" %
%   N9:24  PURIFY_OVERLAP  "STATE Puriify Overlap" %
%   N11:0  PROC_STATE  "STATE The current state of the process" %
%   N9:13  PROC_OVERLAP  "STATE Process Purify Overlap" %
%   N9:21  PURIFY_RUN  "STATE Purify running" %
% Rung: 13 %
% TITLE: TRANSITIONS FOR MANUAL CONTROLS %
SOR XIC B32:0/3 BST CLR N12:0 NXB CLR N12:1 BND EOR
%   B32:0/3  RESET_PURIFIER_CMD %
%   N12:0  PURIFY_STATE  "STATE The current state of the purify process" %
%   N12:1  PURIFY_STATE_BUFFER  "STATE The buffered, previous state of the purify process" %

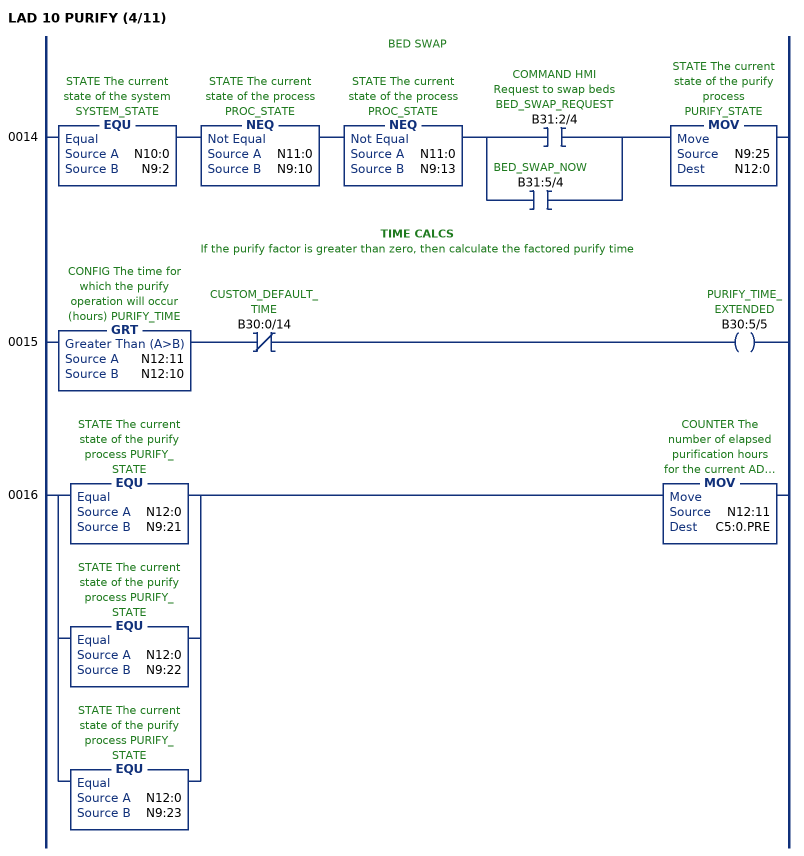
% Rung: 14 %
% BED SWAP %
SOR EQU N10:0 N9:2 NEQ N11:0 N9:10 NEQ N11:0 N9:13 BST XIC B31:2/4 NXB XIC B31:5/4 BND MOV N9:25 N12:0 EOR
%   N10:0  SYSTEM_STATE  "STATE The current state of the system" %
%   N9:2  SYSTEM_PROCESS  "STATE System Process" %
%   N11:0  PROC_STATE  "STATE The current state of the process" %
%   N9:10  PROC_STANDBY  "STATE Process Standby" %
%   N9:13  PROC_OVERLAP  "STATE Process Purify Overlap" %
%   B31:2/4  BED_SWAP_REQUEST  "COMMAND HMI Request to swap beds" %
%   B31:5/4  BED_SWAP_NOW %
%   N9:25  PURIFY_DONE %
%   N12:0  PURIFY_STATE  "STATE The current state of the purify process" %
% Rung: 15 %
% TITLE: TIME CALCS %
% If the purify factor is greater than zero, then calculate the factored purify time %
SOR GRT N12:11 N12:10 XIO B30:0/14 OTE B30:5/5 EOR
%   N12:11  PURIFY_TIME  "CONFIG The time for which the purify operation will occur (hours)" %
%   N12:10  DEFAULT_PURIFY_TIME  "CONFIG The percent output requested by the operator (percent)" %
%   B30:0/14  CUSTOM_DEFAULT_TIME %
%   B30:5/5  PURIFY_TIME_EXTENDED %
% Rung: 16 %
SOR BST EQU N12:0 N9:21 NXB EQU N12:0 N9:22 NXB EQU N12:0 N9:23 BND MOV N12:11 C5:0.PRE EOR
%   N12:0  PURIFY_STATE  "STATE The current state of the purify process" %
%   N9:21  PURIFY_RUN  "STATE Purify running" %
%   N9:22  PURIFY_HOLD  "STATE Purify Hold" %
%   N9:23  PURIFY_MANUAL_HOLD  "STATE Purify Manual Hold" %
%   N12:11  PURIFY_TIME  "CONFIG The time for which the purify operation will occur (hours)" %
%   C5:0  PURIFY_ACTIVE_HOURS  "COUNTER The number of elapsed purification hours for the current ADS" %

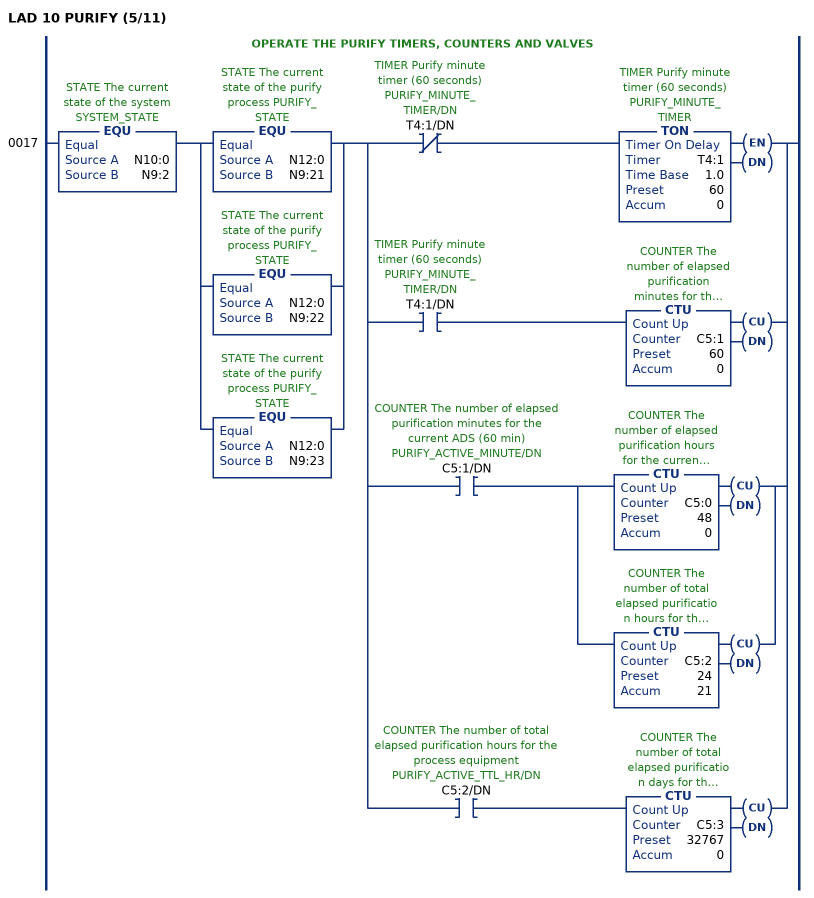
% Rung: 17 %
% TITLE: OPERATE THE PURIFY TIMERS, COUNTERS AND VALVES %
SOR EQU N10:0 N9:2 BST EQU N12:0 N9:21 NXB EQU N12:0 N9:22 NXB EQU N12:0 N9:23 BND BST XIO T4:1/DN TON T4:1 1.0 60 0 NXB XIC T4:1/DN CTU C5:1 60 0 NXB XIC C5:1/DN BST CTU C5:0 48 0 NXB CTU C5:2 24 21 BND NXB XIC C5:2/DN CTU C5:3 32767 0 BND EOR
%   N10:0  SYSTEM_STATE  "STATE The current state of the system" %
%   N9:2  SYSTEM_PROCESS  "STATE System Process" %
%   N12:0  PURIFY_STATE  "STATE The current state of the purify process" %
%   N9:21  PURIFY_RUN  "STATE Purify running" %
%   N9:22  PURIFY_HOLD  "STATE Purify Hold" %
%   N9:23  PURIFY_MANUAL_HOLD  "STATE Purify Manual Hold" %
%   T4:1  PURIFY_MINUTE_TIMER  "TIMER Purify minute timer (60 seconds)" %
%   C5:1  PURIFY_ACTIVE_MINUTE  "COUNTER The number of elapsed purification minutes for the current ADS (60 min)" %
%   C5:0  PURIFY_ACTIVE_HOURS  "COUNTER The number of elapsed purification hours for the current ADS" %
%   C5:2  PURIFY_ACTIVE_TTL_HR  "COUNTER The number of total elapsed purification hours for the process equipment" %
%   C5:3  PURIFY_ACTIVE_TTL_DY  "COUNTER The number of total elapsed purification days for the process equipment" %

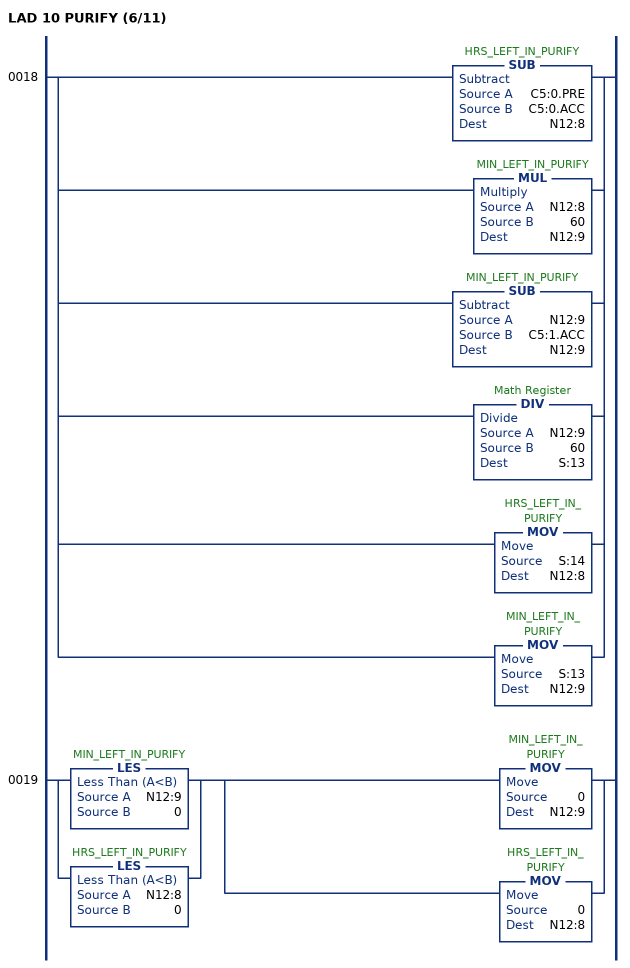
% Rung: 18 %
SOR BST SUB C5:0.PRE C5:0.ACC N12:8 NXB MUL N12:8 60 N12:9 NXB SUB N12:9 C5:1.ACC N12:9 NXB DIV N12:9 60 S:13 NXB MOV S:14 N12:8 NXB MOV S:13 N12:9 BND EOR
%   C5:0  PURIFY_ACTIVE_HOURS  "COUNTER The number of elapsed purification hours for the current ADS" %
%   N12:8  HRS_LEFT_IN_PURIFY %
%   N12:9  MIN_LEFT_IN_PURIFY %
%   C5:1  PURIFY_ACTIVE_MINUTE  "COUNTER The number of elapsed purification minutes for the current ADS (60 min)" %
%   S:13  "Math Register" %
%   S:14  "Math Register" %
% Rung: 19 %
SOR BST LES N12:9 0 NXB LES N12:8 0 BND BST MOV 0 N12:9 NXB MOV 0 N12:8 BND EOR
%   N12:9  MIN_LEFT_IN_PURIFY %
%   N12:8  HRS_LEFT_IN_PURIFY %

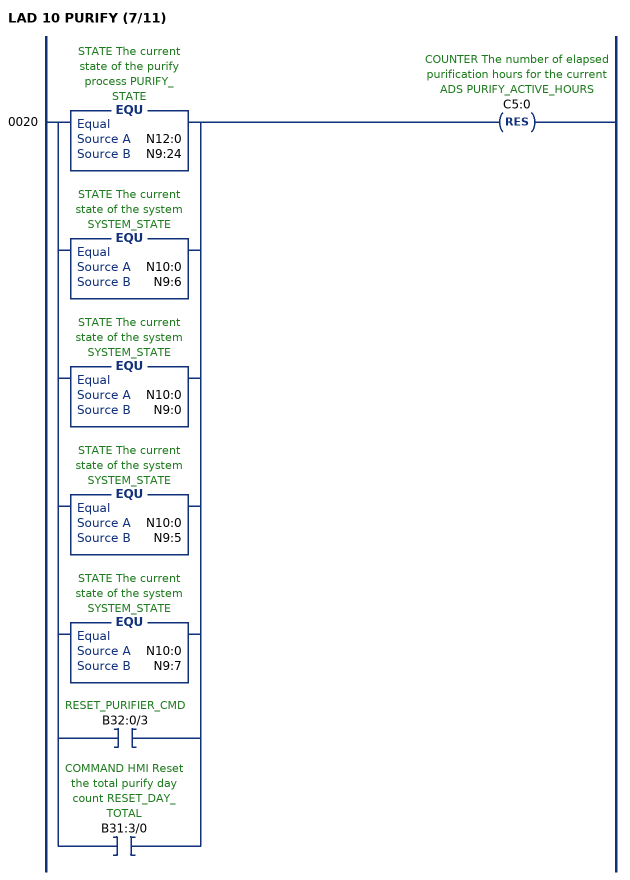
% Rung: 20 %
SOR BST EQU N12:0 N9:24 NXB EQU N10:0 N9:6 NXB EQU N10:0 N9:0 NXB EQU N10:0 N9:5 NXB EQU N10:0 N9:7 NXB XIC B32:0/3 NXB XIC B31:3/0 BND RES C5:0 EOR
%   N12:0  PURIFY_STATE  "STATE The current state of the purify process" %
%   N9:24  PURIFY_OVERLAP  "STATE Puriify Overlap" %
%   N10:0  SYSTEM_STATE  "STATE The current state of the system" %
%   N9:6  SYSTEM_PURGE %
%   N9:0  SYSTEM_OFFLINE %
%   N9:5  SYSTEM_QUICK_START %
%   N9:7  SYSTEM_COLD_START %
%   B32:0/3  RESET_PURIFIER_CMD %
%   B31:3/0  RESET_DAY_TOTAL  "COMMAND HMI Reset the total purify day count" %
%   C5:0  PURIFY_ACTIVE_HOURS  "COUNTER The number of elapsed purification hours for the current ADS" %

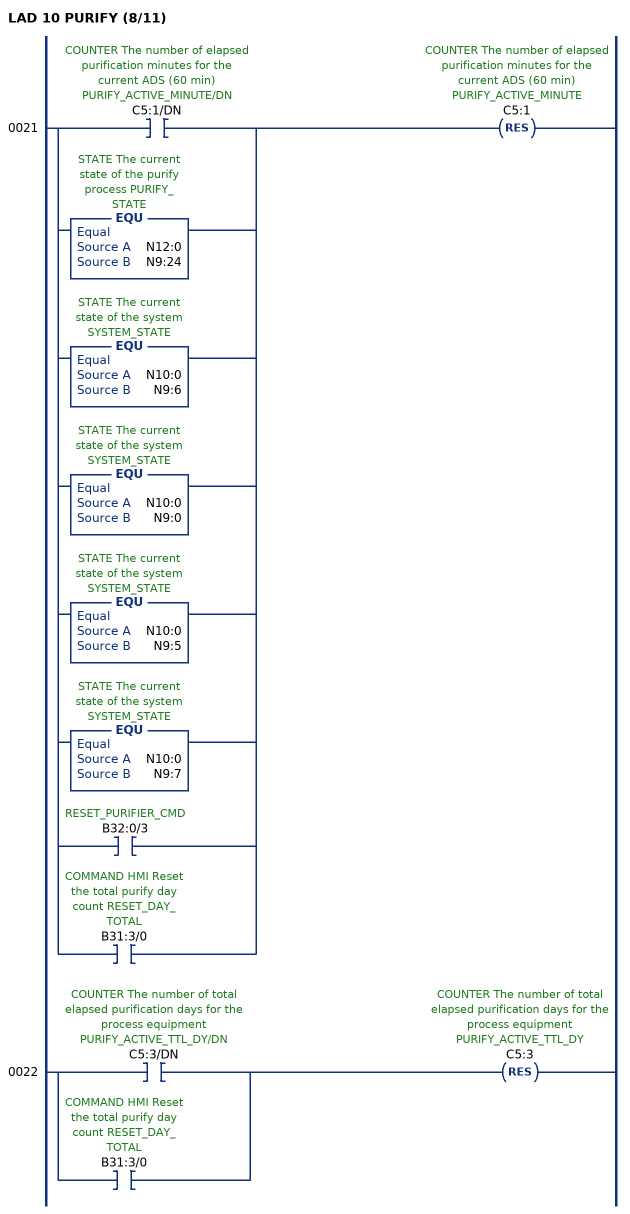
% Rung: 21 %
SOR BST XIC C5:1/DN NXB EQU N12:0 N9:24 NXB EQU N10:0 N9:6 NXB EQU N10:0 N9:0 NXB EQU N10:0 N9:5 NXB EQU N10:0 N9:7 NXB XIC B32:0/3 NXB XIC B31:3/0 BND RES C5:1 EOR
%   C5:1  PURIFY_ACTIVE_MINUTE  "COUNTER The number of elapsed purification minutes for the current ADS (60 min)" %
%   N12:0  PURIFY_STATE  "STATE The current state of the purify process" %
%   N9:24  PURIFY_OVERLAP  "STATE Puriify Overlap" %
%   N10:0  SYSTEM_STATE  "STATE The current state of the system" %
%   N9:6  SYSTEM_PURGE %
%   N9:0  SYSTEM_OFFLINE %
%   N9:5  SYSTEM_QUICK_START %
%   N9:7  SYSTEM_COLD_START %
%   B32:0/3  RESET_PURIFIER_CMD %
%   B31:3/0  RESET_DAY_TOTAL  "COMMAND HMI Reset the total purify day count" %
% Rung: 22 %
SOR BST XIC C5:3/DN NXB XIC B31:3/0 BND RES C5:3 EOR
%   C5:3  PURIFY_ACTIVE_TTL_DY  "COUNTER The number of total elapsed purification days for the process equipment" %
%   B31:3/0  RESET_DAY_TOTAL  "COMMAND HMI Reset the total purify day count" %

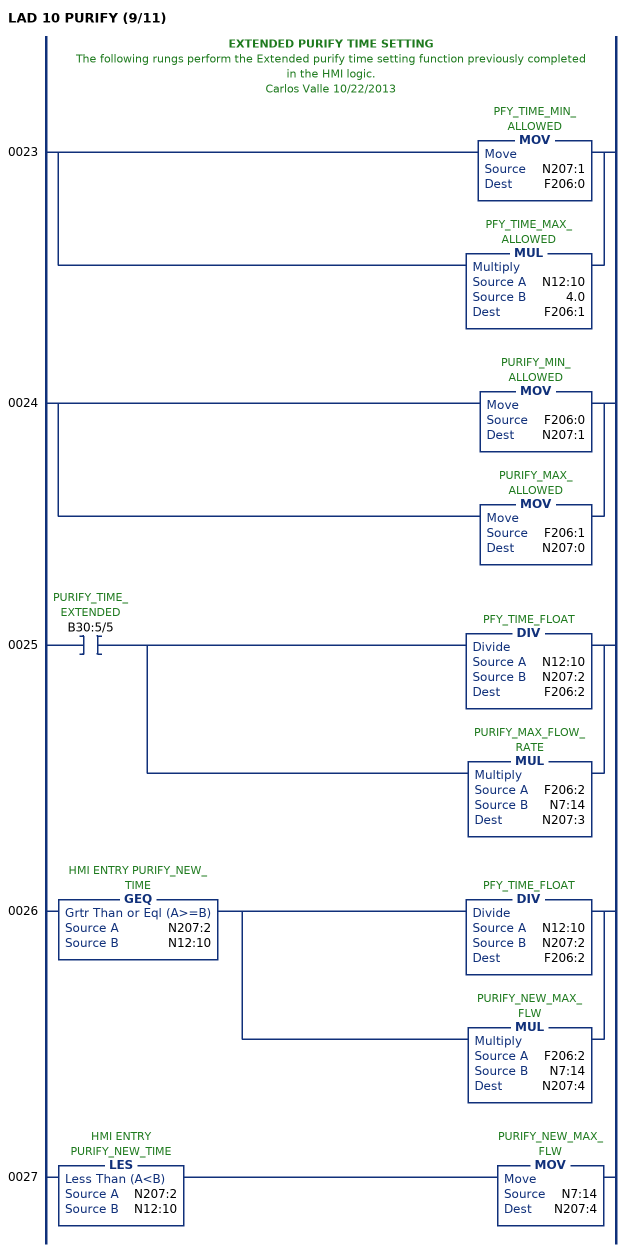
% Rung: 23 %
% TITLE: EXTENDED PURIFY TIME SETTING %
% The following rungs perform the Extended purify time setting function previously completed in the HMI logic.
% Carlos Valle 10/22/2013 %
SOR BST MOV N207:1 F206:0 NXB MUL N12:10 4.0 F206:1 BND EOR
%   N207:1  PURIFY_MIN_ALLOWED %
%   F206:0  PFY_TIME_MIN_ALLOWED %
%   N12:10  DEFAULT_PURIFY_TIME  "CONFIG The percent output requested by the operator (percent)" %
%   F206:1  PFY_TIME_MAX_ALLOWED %
% Rung: 24 %
SOR BST MOV F206:0 N207:1 NXB MOV F206:1 N207:0 BND EOR
%   F206:0  PFY_TIME_MIN_ALLOWED %
%   N207:1  PURIFY_MIN_ALLOWED %
%   F206:1  PFY_TIME_MAX_ALLOWED %
%   N207:0  PURIFY_MAX_ALLOWED %
% Rung: 25 %
SOR XIC B30:5/5 BST DIV N12:10 N207:2 F206:2 NXB MUL F206:2 N7:14 N207:3 BND EOR
%   B30:5/5  PURIFY_TIME_EXTENDED %
%   N12:10  DEFAULT_PURIFY_TIME  "CONFIG The percent output requested by the operator (percent)" %
%   N207:2  PURIFY_NEW_TIME  "HMI ENTRY" %
%   F206:2  PFY_TIME_FLOAT %
%   N7:14  PURIFIER_SIZE %
%   N207:3  PURIFY_MAX_FLOW_RATE %
% Rung: 26 %
SOR GEQ N207:2 N12:10 BST DIV N12:10 N207:2 F206:2 NXB MUL F206:2 N7:14 N207:4 BND EOR
%   N207:2  PURIFY_NEW_TIME  "HMI ENTRY" %
%   N12:10  DEFAULT_PURIFY_TIME  "CONFIG The percent output requested by the operator (percent)" %
%   F206:2  PFY_TIME_FLOAT %
%   N7:14  PURIFIER_SIZE %
%   N207:4  PURIFY_NEW_MAX_FLW %
% Rung: 27 %
SOR LES N207:2 N12:10 MOV N7:14 N207:4 EOR
%   N207:2  PURIFY_NEW_TIME  "HMI ENTRY" %
%   N12:10  DEFAULT_PURIFY_TIME  "CONFIG The percent output requested by the operator (percent)" %
%   N7:14  PURIFIER_SIZE %
%   N207:4  PURIFY_NEW_MAX_FLW %

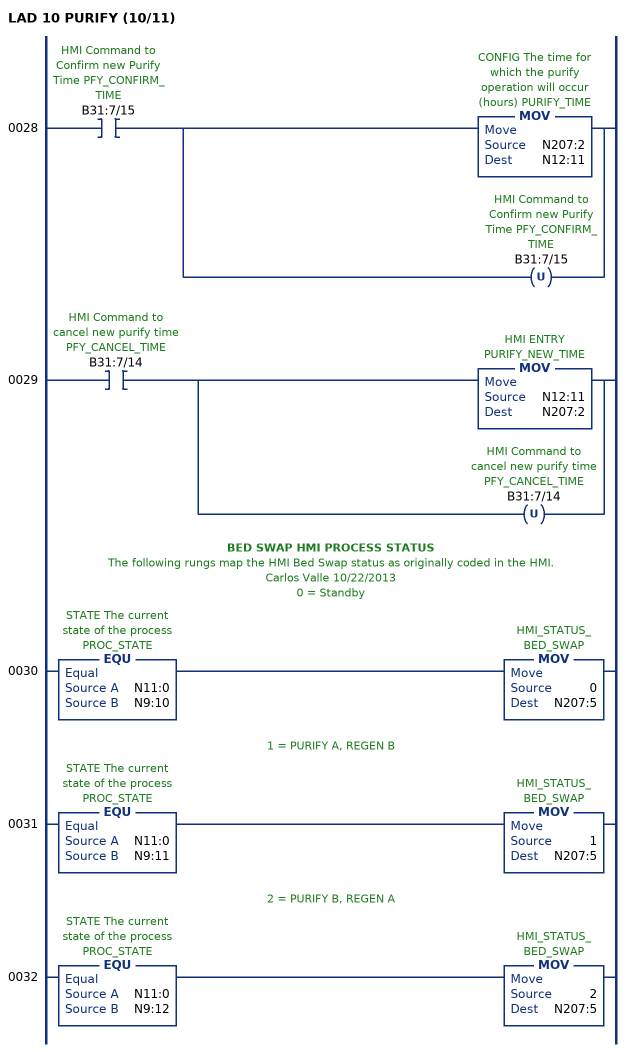
% Rung: 28 %
SOR XIC B31:7/15 BST MOV N207:2 N12:11 NXB OTU B31:7/15 BND EOR
%   B31:7/15  PFY_CONFIRM_TIME  "HMI Command to Confirm new Purify Time" %
%   N207:2  PURIFY_NEW_TIME  "HMI ENTRY" %
%   N12:11  PURIFY_TIME  "CONFIG The time for which the purify operation will occur (hours)" %
% Rung: 29 %
SOR XIC B31:7/14 BST MOV N12:11 N207:2 NXB OTU B31:7/14 BND EOR
%   B31:7/14  PFY_CANCEL_TIME  "HMI Command to cancel new purify time" %
%   N12:11  PURIFY_TIME  "CONFIG The time for which the purify operation will occur (hours)" %
%   N207:2  PURIFY_NEW_TIME  "HMI ENTRY" %
% Rung: 30 %
% TITLE: BED SWAP HMI PROCESS STATUS %
% The following rungs map the HMI Bed Swap status as originally coded in the HMI.
% Carlos Valle 10/22/2013
% 0 = Standby %
SOR EQU N11:0 N9:10 MOV 0 N207:5 EOR
%   N11:0  PROC_STATE  "STATE The current state of the process" %
%   N9:10  PROC_STANDBY  "STATE Process Standby" %
%   N207:5  HMI_STATUS_BED_SWAP %
% Rung: 31 %
% 1 = PURIFY A, REGEN B %
SOR EQU N11:0 N9:11 MOV 1 N207:5 EOR
%   N11:0  PROC_STATE  "STATE The current state of the process" %
%   N9:11  PROC_PFY_A_REG_B  "STATE Process Purify A" %
%   N207:5  HMI_STATUS_BED_SWAP %
% Rung: 32 %
% 2 = PURIFY B, REGEN A %
SOR EQU N11:0 N9:12 MOV 2 N207:5 EOR
%   N11:0  PROC_STATE  "STATE The current state of the process" %
%   N9:12  PROC_PFY_B_REG_A  "STATE Process Purify B" %
%   N207:5  HMI_STATUS_BED_SWAP %

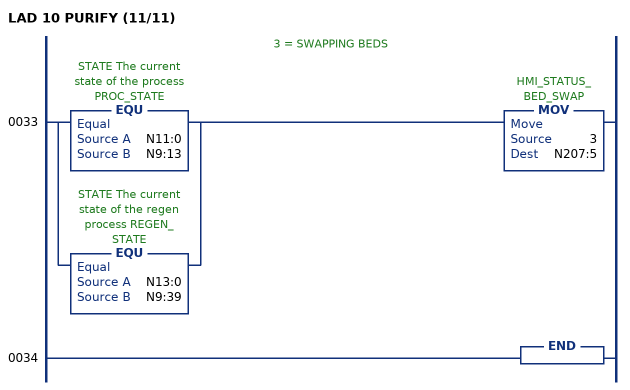
% Rung: 33 %
% 3 = SWAPPING BEDS %
SOR BST EQU N11:0 N9:13 NXB EQU N13:0 N9:39 BND MOV 3 N207:5 EOR
%   N11:0  PROC_STATE  "STATE The current state of the process" %
%   N9:13  PROC_OVERLAP  "STATE Process Purify Overlap" %
%   N13:0  REGEN_STATE  "STATE The current state of the regen process" %
%   N9:39  REGEN_BACKFILL %
%   N207:5  HMI_STATUS_BED_SWAP %
% Rung: 34 %
SOR END EOR

LADDER 11 "REGEN"    % Operates the regen control %
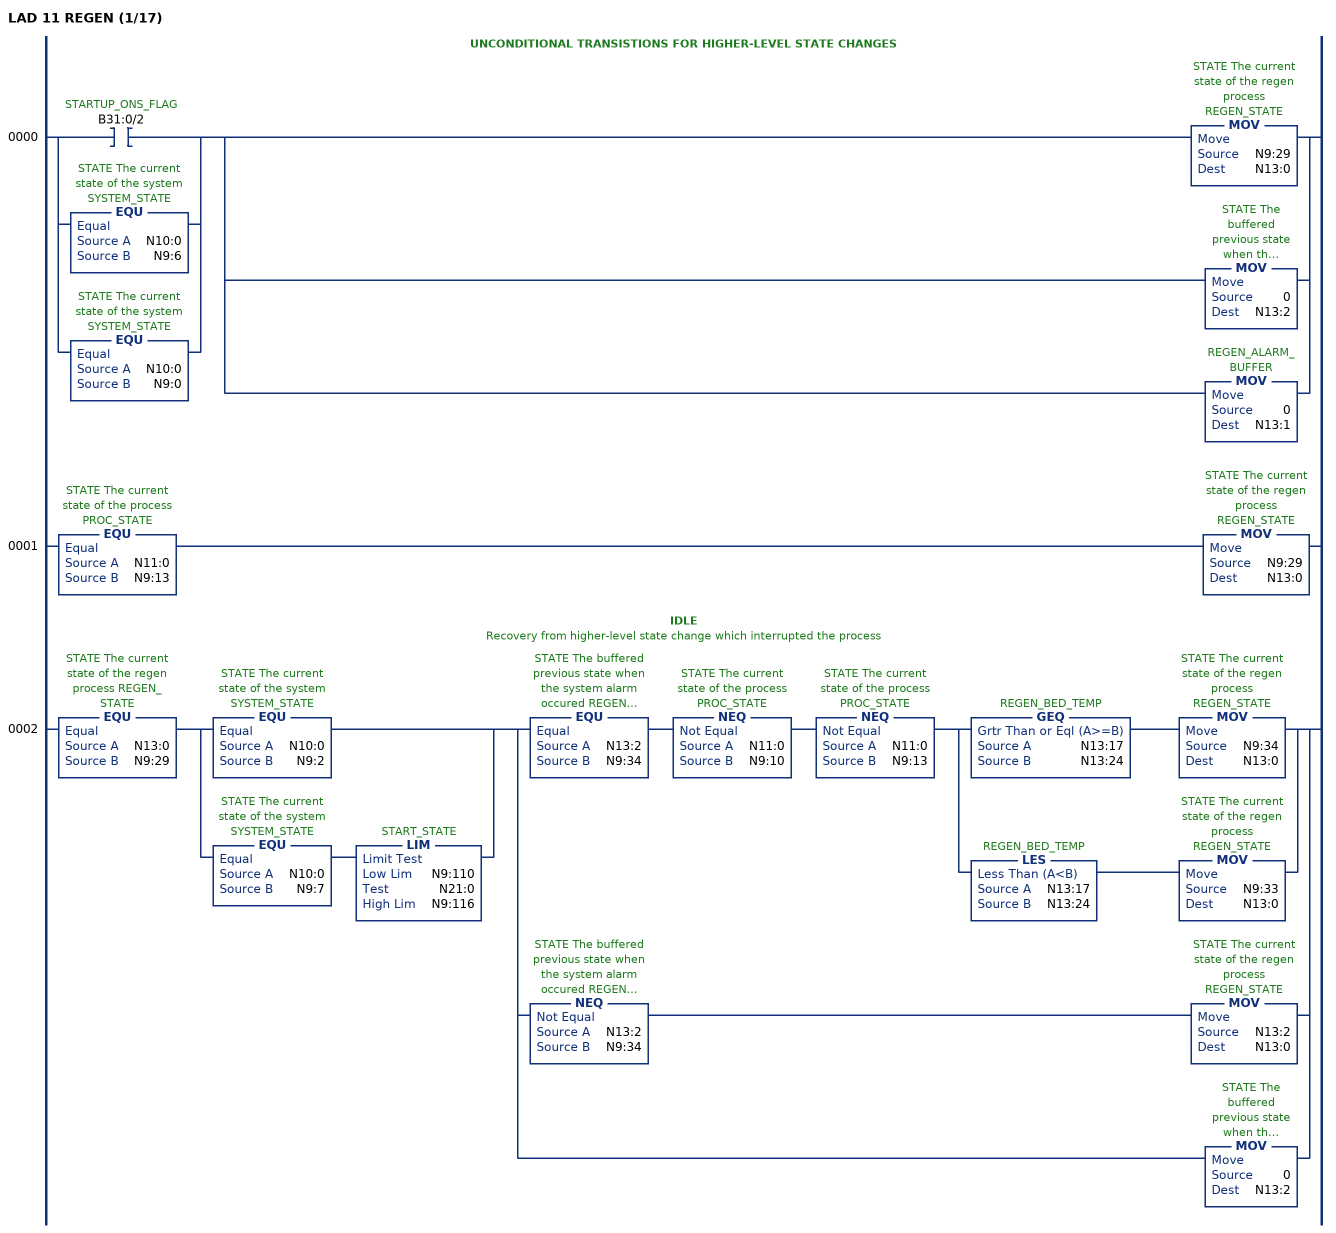
% Rung: 0 %
% TITLE: UNCONDITIONAL TRANSISTIONS FOR HIGHER-LEVEL STATE CHANGES %
SOR BST XIC B31:0/2 NXB EQU N10:0 N9:6 NXB EQU N10:0 N9:0 BND BST MOV N9:29 N13:0 NXB MOV 0 N13:2 NXB MOV 0 N13:1 BND EOR
%   B31:0/2  STARTUP_ONS_FLAG %
%   N10:0  SYSTEM_STATE  "STATE The current state of the system" %
%   N9:6  SYSTEM_PURGE %
%   N9:0  SYSTEM_OFFLINE %
%   N9:29  REGEN_IDLE %
%   N13:0  REGEN_STATE  "STATE The current state of the regen process" %
%   N13:2  REGEN_SYSTEM_BUFFER  "STATE The buffered previous state when the system alarm occured" %
%   N13:1  REGEN_ALARM_BUFFER %
% Rung: 1 %
SOR EQU N11:0 N9:13 MOV N9:29 N13:0 EOR
%   N11:0  PROC_STATE  "STATE The current state of the process" %
%   N9:13  PROC_OVERLAP  "STATE Process Purify Overlap" %
%   N9:29  REGEN_IDLE %
%   N13:0  REGEN_STATE  "STATE The current state of the regen process" %
% Rung: 2 %
% TITLE: IDLE %
% Recovery from higher-level state change which interrupted the process %
SOR EQU N13:0 N9:29 BST EQU N10:0 N9:2 NXB EQU N10:0 N9:7 LIM N9:110 N21:0 N9:116 BND BST EQU N13:2 N9:34 NEQ N11:0 N9:10 NEQ N11:0 N9:13 BST GEQ N13:17 N13:24 MOV N9:34 N13:0 NXB LES N13:17 N13:24 MOV N9:33 N13:0 BND NXB NEQ N13:2 N9:34 MOV N13:2 N13:0 NXB MOV 0 N13:2 BND EOR
%   N13:0  REGEN_STATE  "STATE The current state of the regen process" %
%   N9:29  REGEN_IDLE %
%   N10:0  SYSTEM_STATE  "STATE The current state of the system" %
%   N9:2  SYSTEM_PROCESS  "STATE System Process" %
%   N9:7  SYSTEM_COLD_START %
%   N9:110  START_REG_VENT %
%   N21:0  START_STATE %
%   N9:116  START_REG_BACKFILL %
%   N13:2  REGEN_SYSTEM_BUFFER  "STATE The buffered previous state when the system alarm occured" %
%   N9:34  REGEN_RUN  "STATE Regen Running" %
%   N11:0  PROC_STATE  "STATE The current state of the process" %
%   N9:10  PROC_STANDBY  "STATE Process Standby" %
%   N9:13  PROC_OVERLAP  "STATE Process Purify Overlap" %
%   N13:17  REGEN_BED_TEMP %
%   N13:24  ADS_BED_TEMP_HIGH  "CONFIG The temp at which the regen process may continue" %
%   N9:33  REGEN_HEAT_BED  "STATE Regen Heat wall" %

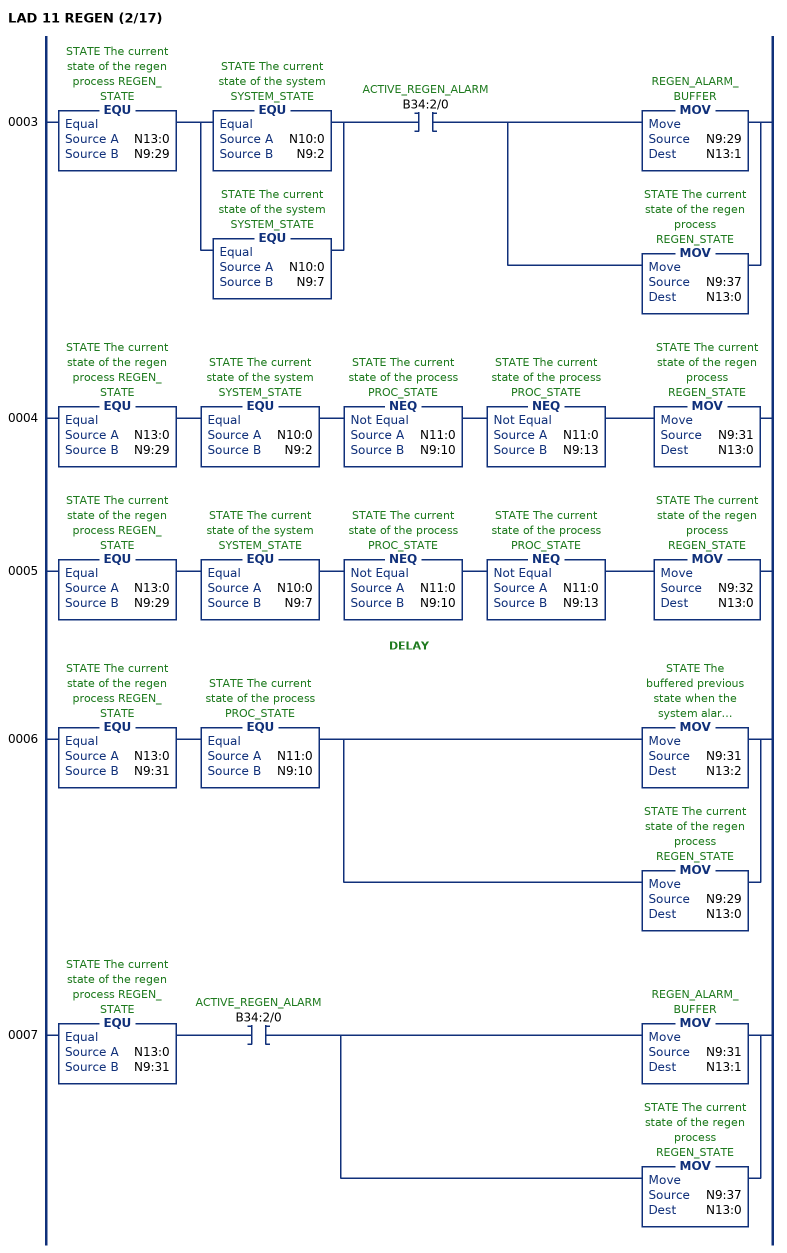
% Rung: 3 %
SOR EQU N13:0 N9:29 BST EQU N10:0 N9:2 NXB EQU N10:0 N9:7 BND XIC B34:2/0 BST MOV N9:29 N13:1 NXB MOV N9:37 N13:0 BND EOR
%   N13:0  REGEN_STATE  "STATE The current state of the regen process" %
%   N9:29  REGEN_IDLE %
%   N10:0  SYSTEM_STATE  "STATE The current state of the system" %
%   N9:2  SYSTEM_PROCESS  "STATE System Process" %
%   N9:7  SYSTEM_COLD_START %
%   B34:2/0  ACTIVE_REGEN_ALARM %
%   N13:1  REGEN_ALARM_BUFFER %
%   N9:37  REGEN_ALARM  "STATE Regen Alarm" %
% Rung: 4 %
SOR EQU N13:0 N9:29 EQU N10:0 N9:2 NEQ N11:0 N9:10 NEQ N11:0 N9:13 MOV N9:31 N13:0 EOR
%   N13:0  REGEN_STATE  "STATE The current state of the regen process" %
%   N9:29  REGEN_IDLE %
%   N10:0  SYSTEM_STATE  "STATE The current state of the system" %
%   N9:2  SYSTEM_PROCESS  "STATE System Process" %
%   N11:0  PROC_STATE  "STATE The current state of the process" %
%   N9:10  PROC_STANDBY  "STATE Process Standby" %
%   N9:13  PROC_OVERLAP  "STATE Process Purify Overlap" %
%   N9:31  REGEN_DELAY  "STATE Regen Delay" %
% Rung: 5 %
SOR EQU N13:0 N9:29 EQU N10:0 N9:7 NEQ N11:0 N9:10 NEQ N11:0 N9:13 MOV N9:32 N13:0 EOR
%   N13:0  REGEN_STATE  "STATE The current state of the regen process" %
%   N9:29  REGEN_IDLE %
%   N10:0  SYSTEM_STATE  "STATE The current state of the system" %
%   N9:7  SYSTEM_COLD_START %
%   N11:0  PROC_STATE  "STATE The current state of the process" %
%   N9:10  PROC_STANDBY  "STATE Process Standby" %
%   N9:13  PROC_OVERLAP  "STATE Process Purify Overlap" %
%   N9:32  REGEN_VENT  "STATE Regen Vent" %
% Rung: 6 %
% TITLE: DELAY %
SOR EQU N13:0 N9:31 EQU N11:0 N9:10 BST MOV N9:31 N13:2 NXB MOV N9:29 N13:0 BND EOR
%   N13:0  REGEN_STATE  "STATE The current state of the regen process" %
%   N9:31  REGEN_DELAY  "STATE Regen Delay" %
%   N11:0  PROC_STATE  "STATE The current state of the process" %
%   N9:10  PROC_STANDBY  "STATE Process Standby" %
%   N13:2  REGEN_SYSTEM_BUFFER  "STATE The buffered previous state when the system alarm occured" %
%   N9:29  REGEN_IDLE %
% Rung: 7 %
SOR EQU N13:0 N9:31 XIC B34:2/0 BST MOV N9:31 N13:1 NXB MOV N9:37 N13:0 BND EOR
%   N13:0  REGEN_STATE  "STATE The current state of the regen process" %
%   N9:31  REGEN_DELAY  "STATE Regen Delay" %
%   B34:2/0  ACTIVE_REGEN_ALARM %
%   N13:1  REGEN_ALARM_BUFFER %
%   N9:37  REGEN_ALARM  "STATE Regen Alarm" %

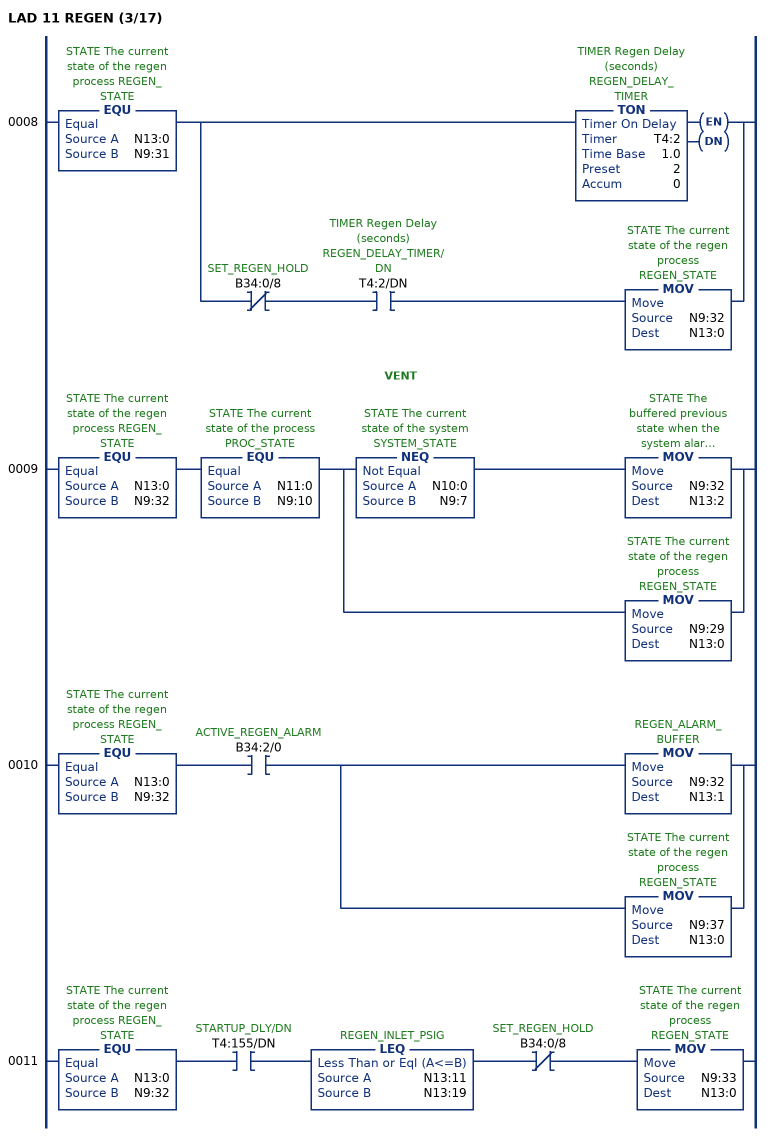
% Rung: 8 %
SOR EQU N13:0 N9:31 BST TON T4:2 1.0 2 0 NXB XIO B34:0/8 XIC T4:2/DN MOV N9:32 N13:0 BND EOR
%   N13:0  REGEN_STATE  "STATE The current state of the regen process" %
%   N9:31  REGEN_DELAY  "STATE Regen Delay" %
%   T4:2  REGEN_DELAY_TIMER  "TIMER Regen Delay (seconds)" %
%   B34:0/8  SET_REGEN_HOLD %
%   N9:32  REGEN_VENT  "STATE Regen Vent" %
% Rung: 9 %
% TITLE: VENT %
SOR EQU N13:0 N9:32 EQU N11:0 N9:10 BST NEQ N10:0 N9:7 MOV N9:32 N13:2 NXB MOV N9:29 N13:0 BND EOR
%   N13:0  REGEN_STATE  "STATE The current state of the regen process" %
%   N9:32  REGEN_VENT  "STATE Regen Vent" %
%   N11:0  PROC_STATE  "STATE The current state of the process" %
%   N9:10  PROC_STANDBY  "STATE Process Standby" %
%   N10:0  SYSTEM_STATE  "STATE The current state of the system" %
%   N9:7  SYSTEM_COLD_START %
%   N13:2  REGEN_SYSTEM_BUFFER  "STATE The buffered previous state when the system alarm occured" %
%   N9:29  REGEN_IDLE %
% Rung: 10 %
SOR EQU N13:0 N9:32 XIC B34:2/0 BST MOV N9:32 N13:1 NXB MOV N9:37 N13:0 BND EOR
%   N13:0  REGEN_STATE  "STATE The current state of the regen process" %
%   N9:32  REGEN_VENT  "STATE Regen Vent" %
%   B34:2/0  ACTIVE_REGEN_ALARM %
%   N13:1  REGEN_ALARM_BUFFER %
%   N9:37  REGEN_ALARM  "STATE Regen Alarm" %
% Rung: 11 %
SOR EQU N13:0 N9:32 XIC T4:155/DN LEQ N13:11 N13:19 XIO B34:0/8 MOV N9:33 N13:0 EOR
%   N13:0  REGEN_STATE  "STATE The current state of the regen process" %
%   N9:32  REGEN_VENT  "STATE Regen Vent" %
%   T4:155  STARTUP_DLY %
%   N13:11  REGEN_INLET_PSIG %
%   N13:19  REGEN_VENT_PRES %
%   B34:0/8  SET_REGEN_HOLD %
%   N9:33  REGEN_HEAT_BED  "STATE Regen Heat wall" %

